	LOCAL CONST Robtarget Tr_meulage_motif_1_P374 :=[[8.13885791015625,-202.05440625,-14.531873046875],[0.696320279376617,-0.571579290814731,-0.275420255163045,0.335527742350052],[0,0,0,0],[8.999999E+09,8.999999E+09,8.999999E+09,8.999999E+09,8.999999E+09,8.999999E+09]];
	LOCAL CONST Robtarget Tr_meulage_motif_1_P375 :=[[8.663193359375,-201.419984375,-15.4485517578125],[0.696320279376617,-0.571579290814731,-0.275420255163045,0.335527742350052],[0,0,0,0],[8.999999E+09,8.999999E+09,8.999999E+09,8.999999E+09,8.999999E+09,8.999999E+09]];
	LOCAL CONST Robtarget Tr_meulage_motif_1_P376 :=[[9.0439765625,-200.94025,-15.87097265625],[0.696320279376617,-0.571579290814731,-0.275420255163045,0.335527742350052],[0,0,0,0],[8.999999E+09,8.999999E+09,8.999999E+09,8.999999E+09,8.999999E+09,8.999999E+09]];
	LOCAL CONST Robtarget Tr_meulage_motif_1_P377 :=[[9.7377255859375,-200.04753125,-16.400830078125],[0.696320279376617,-0.571579290814731,-0.275420255163045,0.335527742350052],[0,0,0,0],[8.999999E+09,8.999999E+09,8.999999E+09,8.999999E+09,8.999999E+09,8.999999E+09]];
	LOCAL CONST Robtarget Tr_meulage_motif_1_P378 :=[[10.2514345703125,-199.37646875,-16.66463671875],[0.696320279376617,-0.571579290814731,-0.275420255163045,0.335527742350052],[0,0,0,0],[8.999999E+09,8.999999E+09,8.999999E+09,8.999999E+09,8.999999E+09,8.999999E+09]];
	LOCAL CONST Robtarget Tr_meulage_motif_1_P379 :=[[10.8147724609375,-198.633921875,-16.868880859375],[0.696320279376617,-0.571579290814731,-0.275420255163045,0.335527742350052],[0,0,0,0],[8.999999E+09,8.999999E+09,8.999999E+09,8.999999E+09,8.999999E+09,8.999999E+09]];
	LOCAL CONST Robtarget Tr_meulage_motif_1_P380 :=[[11.4040810546875,-197.848921875,-16.977291015625],[0.696320279376617,-0.571579290814731,-0.275420255163045,0.335527742350052],[0,0,0,0],[8.999999E+09,8.999999E+09,8.999999E+09,8.999999E+09,8.999999E+09,8.999999E+09]];
	LOCAL CONST Robtarget Tr_meulage_motif_1_P381 :=[[12.000025390625,-197.05515625,-17.087759765625],[0.696320279376617,-0.571579290814731,-0.275420255163045,0.335527742350052],[0,0,0,0],[8.999999E+09,8.999999E+09,8.999999E+09,8.999999E+09,8.999999E+09,8.999999E+09]];
	LOCAL CONST Robtarget Tr_meulage_motif_1_P382 :=[[12.596275390625,-196.252359375,-17.087740234375],[0.696320279376617,-0.571579290814731,-0.275420255163045,0.335527742350052],[0,0,0,0],[8.999999E+09,8.999999E+09,8.999999E+09,8.999999E+09,8.999999E+09,8.999999E+09]];
	LOCAL CONST Robtarget Tr_meulage_motif_1_P383 :=[[13.192525390625,-195.4495625,-17.087720703125],[0.696320279376617,-0.571579290814731,-0.275420255163045,0.335527742350052],[0,0,0,0],[8.999999E+09,8.999999E+09,8.999999E+09,8.999999E+09,8.999999E+09,8.999999E+09]];
	LOCAL CONST Robtarget Tr_meulage_motif_1_P384 :=[[13.7887763671875,-194.646765625,-17.08769921875],[0.696320279376617,-0.571579290814731,-0.275420255163045,0.335527742350052],[0,0,0,0],[8.999999E+09,8.999999E+09,8.999999E+09,8.999999E+09,8.999999E+09,8.999999E+09]];
	LOCAL CONST Robtarget Tr_meulage_motif_1_P385 :=[[14.3850263671875,-193.84396875,-17.0876796875],[0.696320279376617,-0.571579290814731,-0.275420255163045,0.335527742350052],[0,0,0,0],[8.999999E+09,8.999999E+09,8.999999E+09,8.999999E+09,8.999999E+09,8.999999E+09]];
	LOCAL CONST Robtarget Tr_meulage_motif_1_P386 :=[[14.9812763671875,-193.041171875,-17.08766015625],[0.696320279376617,-0.571579290814731,-0.275420255163045,0.335527742350052],[0,0,0,0],[8.999999E+09,8.999999E+09,8.999999E+09,8.999999E+09,8.999999E+09,8.999999E+09]];
	LOCAL CONST Robtarget Tr_meulage_motif_1_P387 :=[[15.57752734375,-192.238375,-17.087638671875],[0.696320279376617,-0.571579290814731,-0.275420255163045,0.335527742350052],[0,0,0,0],[8.999999E+09,8.999999E+09,8.999999E+09,8.999999E+09,8.999999E+09,8.999999E+09]];
	LOCAL CONST Robtarget Tr_meulage_motif_1_P388 :=[[16.17377734375,-191.435578125,-17.087619140625],[0.696320279376617,-0.571579290814731,-0.275420255163045,0.335527742350052],[0,0,0,0],[8.999999E+09,8.999999E+09,8.999999E+09,8.999999E+09,8.999999E+09,8.999999E+09]];
	LOCAL CONST Robtarget Tr_meulage_motif_1_P389 :=[[16.77002734375,-190.632765625,-17.08759765625],[0.696320279376617,-0.571579290814731,-0.275420255163045,0.335527742350052],[0,0,0,0],[8.999999E+09,8.999999E+09,8.999999E+09,8.999999E+09,8.999999E+09,8.999999E+09]];
	LOCAL CONST Robtarget Tr_meulage_motif_1_P390 :=[[17.36627734375,-189.82996875,-17.087578125],[0.696320279376617,-0.571579290814731,-0.275420255163045,0.335527742350052],[0,0,0,0],[8.999999E+09,8.999999E+09,8.999999E+09,8.999999E+09,8.999999E+09,8.999999E+09]];
	LOCAL CONST Robtarget Tr_meulage_motif_1_P391 :=[[17.96252734375,-189.027171875,-17.08755859375],[0.696320279376617,-0.571579290814731,-0.275420255163045,0.335527742350052],[0,0,0,0],[8.999999E+09,8.999999E+09,8.999999E+09,8.999999E+09,8.999999E+09,8.999999E+09]];
	LOCAL CONST Robtarget Tr_meulage_motif_1_P392 :=[[18.558779296875,-188.224375,-17.087537109375],[0.696320279376617,-0.571579290814731,-0.275420255163045,0.335527742350052],[0,0,0,0],[8.999999E+09,8.999999E+09,8.999999E+09,8.999999E+09,8.999999E+09,8.999999E+09]];
	LOCAL CONST Robtarget Tr_meulage_motif_1_P393 :=[[19.155029296875,-187.421578125,-17.087517578125],[0.696320279376617,-0.571579290814731,-0.275420255163045,0.335527742350052],[0,0,0,0],[8.999999E+09,8.999999E+09,8.999999E+09,8.999999E+09,8.999999E+09,8.999999E+09]];
	LOCAL CONST Robtarget Tr_meulage_motif_1_P394 :=[[19.751279296875,-186.61878125,-17.087498046875],[0.696320279376617,-0.571579290814731,-0.275420255163045,0.335527742350052],[0,0,0,0],[8.999999E+09,8.999999E+09,8.999999E+09,8.999999E+09,8.999999E+09,8.999999E+09]];
	LOCAL CONST Robtarget Tr_meulage_motif_1_P395 :=[[20.347529296875,-185.815984375,-17.0874765625],[0.696320279376617,-0.571579290814731,-0.275420255163045,0.335527742350052],[0,0,0,0],[8.999999E+09,8.999999E+09,8.999999E+09,8.999999E+09,8.999999E+09,8.999999E+09]];
	LOCAL CONST Robtarget Tr_meulage_motif_1_P396 :=[[20.943779296875,-185.0131875,-17.08745703125],[0.696320279376617,-0.571579290814731,-0.275420255163045,0.335527742350052],[0,0,0,0],[8.999999E+09,8.999999E+09,8.999999E+09,8.999999E+09,8.999999E+09,8.999999E+09]];
	LOCAL CONST Robtarget Tr_meulage_motif_1_P397 :=[[21.540029296875,-184.210390625,-17.087435546875],[0.696320279376617,-0.571579290814731,-0.275420255163045,0.335527742350052],[0,0,0,0],[8.999999E+09,8.999999E+09,8.999999E+09,8.999999E+09,8.999999E+09,8.999999E+09]];
	LOCAL CONST Robtarget Tr_meulage_motif_1_P398 :=[[22.136279296875,-183.407578125,-17.087416015625],[0.696320279376617,-0.571579290814731,-0.275420255163045,0.335527742350052],[0,0,0,0],[8.999999E+09,8.999999E+09,8.999999E+09,8.999999E+09,8.999999E+09,8.999999E+09]];
	LOCAL CONST Robtarget Tr_meulage_motif_1_P399 :=[[22.73253125,-182.60478125,-17.087396484375],[0.696320279376617,-0.571579290814731,-0.275420255163045,0.335527742350052],[0,0,0,0],[8.999999E+09,8.999999E+09,8.999999E+09,8.999999E+09,8.999999E+09,8.999999E+09]];
	LOCAL CONST Robtarget Tr_meulage_motif_1_P400 :=[[23.32878125,-181.801984375,-17.087375],[0.696320279376617,-0.571579290814731,-0.275420255163045,0.335527742350052],[0,0,0,0],[8.999999E+09,8.999999E+09,8.999999E+09,8.999999E+09,8.999999E+09,8.999999E+09]];
	LOCAL CONST Robtarget Tr_meulage_motif_1_P401 :=[[23.92503125,-180.9991875,-17.08735546875],[0.696320279376617,-0.571579290814731,-0.275420255163045,0.335527742350052],[0,0,0,0],[8.999999E+09,8.999999E+09,8.999999E+09,8.999999E+09,8.999999E+09,8.999999E+09]];
	LOCAL CONST Robtarget Tr_meulage_motif_1_P402 :=[[24.52128125,-180.196390625,-17.0873359375],[0.696320279376617,-0.571579290814731,-0.275420255163045,0.335527742350052],[0,0,0,0],[8.999999E+09,8.999999E+09,8.999999E+09,8.999999E+09,8.999999E+09,8.999999E+09]];
	LOCAL CONST Robtarget Tr_meulage_motif_1_P403 :=[[25.11753125,-179.39359375,-17.087314453125],[0.696320279376617,-0.571579290814731,-0.275420255163045,0.335527742350052],[0,0,0,0],[8.999999E+09,8.999999E+09,8.999999E+09,8.999999E+09,8.999999E+09,8.999999E+09]];
	LOCAL CONST Robtarget Tr_meulage_motif_1_P404 :=[[25.71378125,-178.590796875,-17.087294921875],[0.696320279376617,-0.571579290814731,-0.275420255163045,0.335527742350052],[0,0,0,0],[8.999999E+09,8.999999E+09,8.999999E+09,8.999999E+09,8.999999E+09,8.999999E+09]];
	LOCAL CONST Robtarget Tr_meulage_motif_1_P405 :=[[26.31003125,-177.788,-17.0872734375],[0.696320279376617,-0.571579290814731,-0.275420255163045,0.335527742350052],[0,0,0,0],[8.999999E+09,8.999999E+09,8.999999E+09,8.999999E+09,8.999999E+09,8.999999E+09]];
	LOCAL CONST Robtarget Tr_meulage_motif_1_P406 :=[[26.906283203125,-176.985203125,-17.08725390625],[0.696320279376617,-0.571579290814731,-0.275420255163045,0.335527742350052],[0,0,0,0],[8.999999E+09,8.999999E+09,8.999999E+09,8.999999E+09,8.999999E+09,8.999999E+09]];
	LOCAL CONST Robtarget Tr_meulage_motif_1_P407 :=[[27.502533203125,-176.18240625,-17.087234375],[0.696320279376617,-0.571579290814731,-0.275420255163045,0.335527742350052],[0,0,0,0],[8.999999E+09,8.999999E+09,8.999999E+09,8.999999E+09,8.999999E+09,8.999999E+09]];
	LOCAL CONST Robtarget Tr_meulage_motif_1_P408 :=[[28.098783203125,-175.37959375,-17.087212890625],[0.696320279376617,-0.571579290814731,-0.275420255163045,0.335527742350052],[0,0,0,0],[8.999999E+09,8.999999E+09,8.999999E+09,8.999999E+09,8.999999E+09,8.999999E+09]];
	LOCAL CONST Robtarget Tr_meulage_motif_1_P409 :=[[28.695033203125,-174.576796875,-17.087193359375],[0.696320279376617,-0.571579290814731,-0.275420255163045,0.335527742350052],[0,0,0,0],[8.999999E+09,8.999999E+09,8.999999E+09,8.999999E+09,8.999999E+09,8.999999E+09]];
	LOCAL CONST Robtarget Tr_meulage_motif_1_P410 :=[[29.291283203125,-173.774,-17.087173828125],[0.696320279376617,-0.571579290814731,-0.275420255163045,0.335527742350052],[0,0,0,0],[8.999999E+09,8.999999E+09,8.999999E+09,8.999999E+09,8.999999E+09,8.999999E+09]];
	LOCAL CONST Robtarget Tr_meulage_motif_1_P411 :=[[29.887533203125,-172.971203125,-17.08715234375],[0.696320279376617,-0.571579290814731,-0.275420255163045,0.335527742350052],[0,0,0,0],[8.999999E+09,8.999999E+09,8.999999E+09,8.999999E+09,8.999999E+09,8.999999E+09]];
	LOCAL CONST Robtarget Tr_meulage_motif_1_P412 :=[[30.48378515625,-172.16840625,-17.0871328125],[0.696320279376617,-0.571579290814731,-0.275420255163045,0.335527742350052],[0,0,0,0],[8.999999E+09,8.999999E+09,8.999999E+09,8.999999E+09,8.999999E+09,8.999999E+09]];
	LOCAL CONST Robtarget Tr_meulage_motif_1_P413 :=[[31.08003515625,-171.365609375,-17.087111328125],[0.696320279376617,-0.571579290814731,-0.275420255163045,0.335527742350052],[0,0,0,0],[8.999999E+09,8.999999E+09,8.999999E+09,8.999999E+09,8.999999E+09,8.999999E+09]];
	LOCAL CONST Robtarget Tr_meulage_motif_1_P414 :=[[31.67628515625,-170.5628125,-17.087091796875],[0.696320279376617,-0.571579290814731,-0.275420255163045,0.335527742350052],[0,0,0,0],[8.999999E+09,8.999999E+09,8.999999E+09,8.999999E+09,8.999999E+09,8.999999E+09]];
	LOCAL CONST Robtarget Tr_meulage_motif_1_P415 :=[[32.27253515625,-169.760015625,-17.087072265625],[0.696320279376617,-0.571579290814731,-0.275420255163045,0.335527742350052],[0,0,0,0],[8.999999E+09,8.999999E+09,8.999999E+09,8.999999E+09,8.999999E+09,8.999999E+09]];
	LOCAL CONST Robtarget Tr_meulage_motif_1_P416 :=[[32.86878515625,-168.95721875,-17.08705078125],[0.696320279376617,-0.571579290814731,-0.275420255163045,0.335527742350052],[0,0,0,0],[8.999999E+09,8.999999E+09,8.999999E+09,8.999999E+09,8.999999E+09,8.999999E+09]];
	LOCAL CONST Robtarget Tr_meulage_motif_1_P417 :=[[33.46503515625,-168.15440625,-17.08703125],[0.696320279376617,-0.571579290814731,-0.275420255163045,0.335527742350052],[0,0,0,0],[8.999999E+09,8.999999E+09,8.999999E+09,8.999999E+09,8.999999E+09,8.999999E+09]];
	LOCAL CONST Robtarget Tr_meulage_motif_1_P418 :=[[34.06128515625,-167.351609375,-17.08701171875],[0.696320279376617,-0.571579290814731,-0.275420255163045,0.335527742350052],[0,0,0,0],[8.999999E+09,8.999999E+09,8.999999E+09,8.999999E+09,8.999999E+09,8.999999E+09]];
	LOCAL CONST Robtarget Tr_meulage_motif_1_P419 :=[[34.65753515625,-166.5488125,-17.086990234375],[0.696320279376617,-0.571579290814731,-0.275420255163045,0.335527742350052],[0,0,0,0],[8.999999E+09,8.999999E+09,8.999999E+09,8.999999E+09,8.999999E+09,8.999999E+09]];
	LOCAL CONST Robtarget Tr_meulage_motif_1_P420 :=[[35.25378515625,-165.746015625,-17.086970703125],[0.696320279376617,-0.571579290814731,-0.275420255163045,0.335527742350052],[0,0,0,0],[8.999999E+09,8.999999E+09,8.999999E+09,8.999999E+09,8.999999E+09,8.999999E+09]];
	LOCAL CONST Robtarget Tr_meulage_motif_1_P421 :=[[35.85003515625,-164.94321875,-17.08694921875],[0.696320279376617,-0.571579290814731,-0.275420255163045,0.335527742350052],[0,0,0,0],[8.999999E+09,8.999999E+09,8.999999E+09,8.999999E+09,8.999999E+09,8.999999E+09]];
	LOCAL CONST Robtarget Tr_meulage_motif_1_P422 :=[[36.4462890625,-164.140421875,-17.0869296875],[0.696320279376617,-0.571579290814731,-0.275420255163045,0.335527742350052],[0,0,0,0],[8.999999E+09,8.999999E+09,8.999999E+09,8.999999E+09,8.999999E+09,8.999999E+09]];
	LOCAL CONST Robtarget Tr_meulage_motif_1_P423 :=[[37.0425390625,-163.337625,-17.08691015625],[0.696320279376617,-0.571579290814731,-0.275420255163045,0.335527742350052],[0,0,0,0],[8.999999E+09,8.999999E+09,8.999999E+09,8.999999E+09,8.999999E+09,8.999999E+09]];
	LOCAL CONST Robtarget Tr_meulage_motif_1_P424 :=[[37.6387890625,-162.534828125,-17.086888671875],[0.696320279376617,-0.571579290814731,-0.275420255163045,0.335527742350052],[0,0,0,0],[8.999999E+09,8.999999E+09,8.999999E+09,8.999999E+09,8.999999E+09,8.999999E+09]];
	LOCAL CONST Robtarget Tr_meulage_motif_1_P425 :=[[38.2350390625,-161.73203125,-17.086869140625],[0.696320279376617,-0.571579290814731,-0.275420255163045,0.335527742350052],[0,0,0,0],[8.999999E+09,8.999999E+09,8.999999E+09,8.999999E+09,8.999999E+09,8.999999E+09]];
	LOCAL CONST Robtarget Tr_meulage_motif_1_P426 :=[[38.8312890625,-160.92921875,-17.086849609375],[0.696320279376617,-0.571579290814731,-0.275420255163045,0.335527742350052],[0,0,0,0],[8.999999E+09,8.999999E+09,8.999999E+09,8.999999E+09,8.999999E+09,8.999999E+09]];
	LOCAL CONST Robtarget Tr_meulage_motif_1_P427 :=[[39.4275390625,-160.126421875,-17.086828125],[0.696320279376617,-0.571579290814731,-0.275420255163045,0.335527742350052],[0,0,0,0],[8.999999E+09,8.999999E+09,8.999999E+09,8.999999E+09,8.999999E+09,8.999999E+09]];
	LOCAL CONST Robtarget Tr_meulage_motif_1_P428 :=[[40.0237890625,-159.323625,-17.08680859375],[0.696320279376617,-0.571579290814731,-0.275420255163045,0.335527742350052],[0,0,0,0],[8.999999E+09,8.999999E+09,8.999999E+09,8.999999E+09,8.999999E+09,8.999999E+09]];
	LOCAL CONST Robtarget Tr_meulage_motif_1_P429 :=[[40.6200390625,-158.520828125,-17.086787109375],[0.696320279376617,-0.571579290814731,-0.275420255163045,0.335527742350052],[0,0,0,0],[8.999999E+09,8.999999E+09,8.999999E+09,8.999999E+09,8.999999E+09,8.999999E+09]];
	LOCAL CONST Robtarget Tr_meulage_motif_1_P430 :=[[41.2162890625,-157.71803125,-17.086767578125],[0.696320279376617,-0.571579290814731,-0.275420255163045,0.335527742350052],[0,0,0,0],[8.999999E+09,8.999999E+09,8.999999E+09,8.999999E+09,8.999999E+09,8.999999E+09]];
	LOCAL CONST Robtarget Tr_meulage_motif_1_P431 :=[[41.8125390625,-156.915234375,-17.086748046875],[0.696320279376617,-0.571579290814731,-0.275420255163045,0.335527742350052],[0,0,0,0],[8.999999E+09,8.999999E+09,8.999999E+09,8.999999E+09,8.999999E+09,8.999999E+09]];
	LOCAL CONST Robtarget Tr_meulage_motif_1_P432 :=[[42.4087890625,-156.1124375,-17.0867265625],[0.696320279376617,-0.571579290814731,-0.275420255163045,0.335527742350052],[0,0,0,0],[8.999999E+09,8.999999E+09,8.999999E+09,8.999999E+09,8.999999E+09,8.999999E+09]];
	LOCAL CONST Robtarget Tr_meulage_motif_1_P433 :=[[43.0050390625,-155.309640625,-17.08670703125],[0.696320279376617,-0.571579290814731,-0.275420255163045,0.335527742350052],[0,0,0,0],[8.999999E+09,8.999999E+09,8.999999E+09,8.999999E+09,8.999999E+09,8.999999E+09]];
	LOCAL CONST Robtarget Tr_meulage_motif_1_P434 :=[[43.6012890625,-154.50684375,-17.0866875],[0.696320279376617,-0.571579290814731,-0.275420255163045,0.335527742350052],[0,0,0,0],[8.999999E+09,8.999999E+09,8.999999E+09,8.999999E+09,8.999999E+09,8.999999E+09]];
	LOCAL CONST Robtarget Tr_meulage_motif_1_degg1 :=[[51.2725174233444,-160.618666051073,-19.0355034471531],[0.696320279376617,-0.571579290814731,-0.275420255163045,0.335527742350052],[0,0,0,0],[8.999999E+09,8.999999E+09,8.999999E+09,8.999999E+09,8.999999E+09,8.999999E+09]];
	LOCAL CONST Robtarget Tr_meulage_motif_1_degg2 :=[[197.025856279388,-276.743289771468,-56.063006443061],[0.696320279376617,-0.571579290814731,-0.275420255163045,0.335527742350052],[0,0,0,0],[8.999999E+09,8.999999E+09,8.999999E+09,8.999999E+09,8.999999E+09,8.999999E+09]];
	LOCAL CONST Robtarget Tr_meulage_motif_2_App1 :=[[79.1385711104323,111.598654466444,-198.295056790946],[3.80360857770028E-05,0.00767312788400758,0.0049568441043783,-0.999958274808633],[0,0,0,0],[8.999999E+09,8.999999E+09,8.999999E+09,8.999999E+09,8.999999E+09,8.999999E+09]];
	LOCAL CONST Robtarget Tr_meulage_motif_2_App2 :=[[76.2229758211466,109.715021395197,-8.32676672504532],[3.80360857770028E-05,0.00767312788400758,0.0049568441043783,-0.999958274808633],[0,0,0,0],[8.999999E+09,8.999999E+09,8.999999E+09,8.999999E+09,8.999999E+09,8.999999E+09]];
	LOCAL CONST Robtarget Tr_meulage_motif_2_P0 :=[[76.0695234375,109.6158828125,1.67156433105469],[3.80360857770028E-05,0.00767312788400758,0.0049568441043783,-0.999958274808633],[0,0,0,0],[8.999999E+09,8.999999E+09,8.999999E+09,8.999999E+09,8.999999E+09,8.999999E+09]];
	LOCAL CONST Robtarget Tr_meulage_motif_2_P1 :=[[75.071609375,109.5513046875,1.67191589355469],[3.80360857770028E-05,0.00767312788400758,0.0049568441043783,-0.999958274808633],[0,0,0,0],[8.999999E+09,8.999999E+09,8.999999E+09,8.999999E+09,8.999999E+09,8.999999E+09]];
	LOCAL CONST Robtarget Tr_meulage_motif_2_P2 :=[[74.0736953125,109.4867265625,1.67226745605469],[3.80360857770028E-05,0.00767312788400758,0.0049568441043783,-0.999958274808633],[0,0,0,0],[8.999999E+09,8.999999E+09,8.999999E+09,8.999999E+09,8.999999E+09,8.999999E+09]];
	LOCAL CONST Robtarget Tr_meulage_motif_2_P3 :=[[73.07578125,109.4221484375,1.67261889648438],[3.80360857770028E-05,0.00767312788400758,0.0049568441043783,-0.999958274808633],[0,0,0,0],[8.999999E+09,8.999999E+09,8.999999E+09,8.999999E+09,8.999999E+09,8.999999E+09]];
	LOCAL CONST Robtarget Tr_meulage_motif_2_P4 :=[[72.0778671875,109.3575703125,1.67297045898438],[3.80360857770028E-05,0.00767312788400758,0.0049568441043783,-0.999958274808633],[0,0,0,0],[8.999999E+09,8.999999E+09,8.999999E+09,8.999999E+09,8.999999E+09,8.999999E+09]];
	LOCAL CONST Robtarget Tr_meulage_motif_2_P5 :=[[71.079953125,109.293,1.67332202148438],[3.80360857770028E-05,0.00767312788400758,0.0049568441043783,-0.999958274808633],[0,0,0,0],[8.999999E+09,8.999999E+09,8.999999E+09,8.999999E+09,8.999999E+09,8.999999E+09]];
	LOCAL CONST Robtarget Tr_meulage_motif_2_P6 :=[[70.082046875,109.228421875,1.67367358398438],[3.80360857770028E-05,0.00767312788400758,0.0049568441043783,-0.999958274808633],[0,0,0,0],[8.999999E+09,8.999999E+09,8.999999E+09,8.999999E+09,8.999999E+09,8.999999E+09]];
	LOCAL CONST Robtarget Tr_meulage_motif_2_P7 :=[[69.0841328125,109.16384375,1.67402514648437],[3.80360857770028E-05,0.00767312788400758,0.0049568441043783,-0.999958274808633],[0,0,0,0],[8.999999E+09,8.999999E+09,8.999999E+09,8.999999E+09,8.999999E+09,8.999999E+09]];
	LOCAL CONST Robtarget Tr_meulage_motif_2_P8 :=[[68.08621875,109.099265625,1.67437670898438],[3.80360857770028E-05,0.00767312788400758,0.0049568441043783,-0.999958274808633],[0,0,0,0],[8.999999E+09,8.999999E+09,8.999999E+09,8.999999E+09,8.999999E+09,8.999999E+09]];
	LOCAL CONST Robtarget Tr_meulage_motif_2_P9 :=[[67.0883046875,109.0346875,1.67472827148437],[3.80360857770028E-05,0.00767312788400758,0.0049568441043783,-0.999958274808633],[0,0,0,0],[8.999999E+09,8.999999E+09,8.999999E+09,8.999999E+09,8.999999E+09,8.999999E+09]];
	LOCAL CONST Robtarget Tr_meulage_motif_2_P10 :=[[66.090390625,108.9701171875,1.67507983398438],[3.80360857770028E-05,0.00767312788400758,0.0049568441043783,-0.999958274808633],[0,0,0,0],[8.999999E+09,8.999999E+09,8.999999E+09,8.999999E+09,8.999999E+09,8.999999E+09]];
	LOCAL CONST Robtarget Tr_meulage_motif_2_P11 :=[[65.09248046875,108.9055390625,1.67543127441406],[3.80360857770028E-05,0.00767312788400758,0.0049568441043783,-0.999958274808633],[0,0,0,0],[8.999999E+09,8.999999E+09,8.999999E+09,8.999999E+09,8.999999E+09,8.999999E+09]];
	LOCAL CONST Robtarget Tr_meulage_motif_2_P12 :=[[64.09456640625,108.8409609375,1.67578283691406],[3.80360857770028E-05,0.00767312788400758,0.0049568441043783,-0.999958274808633],[0,0,0,0],[8.999999E+09,8.999999E+09,8.999999E+09,8.999999E+09,8.999999E+09,8.999999E+09]];
	LOCAL CONST Robtarget Tr_meulage_motif_2_P13 :=[[63.09665625,108.7763828125,1.67613439941406],[3.80360857770028E-05,0.00767312788400758,0.0049568441043783,-0.999958274808633],[0,0,0,0],[8.999999E+09,8.999999E+09,8.999999E+09,8.999999E+09,8.999999E+09,8.999999E+09]];
	LOCAL CONST Robtarget Tr_meulage_motif_2_P14 :=[[62.0987421875,108.7118046875,1.67648596191406],[3.80360857770028E-05,0.00767312788400758,0.0049568441043783,-0.999958274808633],[0,0,0,0],[8.999999E+09,8.999999E+09,8.999999E+09,8.999999E+09,8.999999E+09,8.999999E+09]];
	LOCAL CONST Robtarget Tr_meulage_motif_2_P15 :=[[61.100828125,108.6472265625,1.67683752441406],[3.80360857770028E-05,0.00767312788400758,0.0049568441043783,-0.999958274808633],[0,0,0,0],[8.999999E+09,8.999999E+09,8.999999E+09,8.999999E+09,8.999999E+09,8.999999E+09]];
	LOCAL CONST Robtarget Tr_meulage_motif_2_P16 :=[[60.10291796875,108.58265625,1.67718908691406],[3.80360857770028E-05,0.00767312788400758,0.0049568441043783,-0.999958274808633],[0,0,0,0],[8.999999E+09,8.999999E+09,8.999999E+09,8.999999E+09,8.999999E+09,8.999999E+09]];
	LOCAL CONST Robtarget Tr_meulage_motif_2_P17 :=[[59.10500390625,108.518078125,1.67754064941406],[3.80360857770028E-05,0.00767312788400758,0.0049568441043783,-0.999958274808633],[0,0,0,0],[8.999999E+09,8.999999E+09,8.999999E+09,8.999999E+09,8.999999E+09,8.999999E+09]];
	LOCAL CONST Robtarget Tr_meulage_motif_2_P18 :=[[58.10708984375,108.4535,1.67789221191406],[3.80360857770028E-05,0.00767312788400758,0.0049568441043783,-0.999958274808633],[0,0,0,0],[8.999999E+09,8.999999E+09,8.999999E+09,8.999999E+09,8.999999E+09,8.999999E+09]];
	LOCAL CONST Robtarget Tr_meulage_motif_2_P19 :=[[57.1094609375,108.499765625,1.67763696289063],[3.80360857770028E-05,0.00767312788400758,0.0049568441043783,-0.999958274808633],[0,0,0,0],[8.999999E+09,8.999999E+09,8.999999E+09,8.999999E+09,8.999999E+09,8.999999E+09]];
	LOCAL CONST Robtarget Tr_meulage_motif_2_P20 :=[[56.151296875,108.649390625,1.67681604003906],[3.80360857770028E-05,0.00767312788400758,0.0049568441043783,-0.999958274808633],[0,0,0,0],[8.999999E+09,8.999999E+09,8.999999E+09,8.999999E+09,8.999999E+09,8.999999E+09]];
	LOCAL CONST Robtarget Tr_meulage_motif_2_P21 :=[[55.2828046875,108.86559375,1.675630859375],[3.80360857770028E-05,0.00767312788400758,0.0049568441043783,-0.999958274808633],[0,0,0,0],[8.999999E+09,8.999999E+09,8.999999E+09,8.999999E+09,8.999999E+09,8.999999E+09]];
	LOCAL CONST Robtarget Tr_meulage_motif_2_P22 :=[[54.51661328125,109.0925234375,1.67438720703125],[3.80360857770028E-05,0.00767312788400758,0.0049568441043783,-0.999958274808633],[0,0,0,0],[8.999999E+09,8.999999E+09,8.999999E+09,8.999999E+09,8.999999E+09,8.999999E+09]];
	LOCAL CONST Robtarget Tr_meulage_motif_2_P23 :=[[53.37805859375,109.63625,1.67140869140625],[3.80360857770028E-05,0.00767312788400758,0.0049568441043783,-0.999958274808633],[0,0,0,0],[8.999999E+09,8.999999E+09,8.999999E+09,8.999999E+09,8.999999E+09,8.999999E+09]];
	LOCAL CONST Robtarget Tr_meulage_motif_2_P24 :=[[52.30158203125,110.4160078125,1.66713830566406],[3.80360857770028E-05,0.00767312788400758,0.0049568441043783,-0.999958274808633],[0,0,0,0],[8.999999E+09,8.999999E+09,8.999999E+09,8.999999E+09,8.999999E+09,8.999999E+09]];
	LOCAL CONST Robtarget Tr_meulage_motif_2_P25 :=[[51.38957421875,111.3829921875,1.66184338378906],[3.80360857770028E-05,0.00767312788400758,0.0049568441043783,-0.999958274808633],[0,0,0,0],[8.999999E+09,8.999999E+09,8.999999E+09,8.999999E+09,8.999999E+09,8.999999E+09]];
	LOCAL CONST Robtarget Tr_meulage_motif_2_P26 :=[[50.830359375,112.4653046875,1.65591772460938],[3.80360857770028E-05,0.00767312788400758,0.0049568441043783,-0.999958274808633],[0,0,0,0],[8.999999E+09,8.999999E+09,8.999999E+09,8.999999E+09,8.999999E+09,8.999999E+09]];
	LOCAL CONST Robtarget Tr_meulage_motif_2_P27 :=[[50.75840625,113.1580625,1.65212561035156],[3.80360857770028E-05,0.00767312788400758,0.0049568441043783,-0.999958274808633],[0,0,0,0],[8.999999E+09,8.999999E+09,8.999999E+09,8.999999E+09,8.999999E+09,8.999999E+09]];
	LOCAL CONST Robtarget Tr_meulage_motif_2_P28 :=[[50.71570703125,113.817921875,1.64851342773437],[3.80360857770028E-05,0.00767312788400758,0.0049568441043783,-0.999958274808633],[0,0,0,0],[8.999999E+09,8.999999E+09,8.999999E+09,8.999999E+09,8.999999E+09,8.999999E+09]];
	LOCAL CONST Robtarget Tr_meulage_motif_2_P29 :=[[50.7277734375,114.481171875,1.64488293457031],[3.80360857770028E-05,0.00767312788400758,0.0049568441043783,-0.999958274808633],[0,0,0,0],[8.999999E+09,8.999999E+09,8.999999E+09,8.999999E+09,8.999999E+09,8.999999E+09]];
	LOCAL CONST Robtarget Tr_meulage_motif_2_P30 :=[[51.1538046875,115.61278125,1.638689453125],[3.80360857770028E-05,0.00767312788400758,0.0049568441043783,-0.999958274808633],[0,0,0,0],[8.999999E+09,8.999999E+09,8.999999E+09,8.999999E+09,8.999999E+09,8.999999E+09]];
	LOCAL CONST Robtarget Tr_meulage_motif_2_P31 :=[[51.94363671875,116.672609375,1.6328896484375],[3.80360857770028E-05,0.00767312788400758,0.0049568441043783,-0.999958274808633],[0,0,0,0],[8.999999E+09,8.999999E+09,8.999999E+09,8.999999E+09,8.999999E+09,8.999999E+09]];
	LOCAL CONST Robtarget Tr_meulage_motif_2_P32 :=[[52.91137890625,117.565828125,1.62800207519531],[3.80360857770028E-05,0.00767312788400758,0.0049568441043783,-0.999958274808633],[0,0,0,0],[8.999999E+09,8.999999E+09,8.999999E+09,8.999999E+09,8.999999E+09,8.999999E+09]];
	LOCAL CONST Robtarget Tr_meulage_motif_2_P33 :=[[53.571484375,118.0051171875,1.62559875488281],[3.80360857770028E-05,0.00767312788400758,0.0049568441043783,-0.999958274808633],[0,0,0,0],[8.999999E+09,8.999999E+09,8.999999E+09,8.999999E+09,8.999999E+09,8.999999E+09]];
	LOCAL CONST Robtarget Tr_meulage_motif_2_P34 :=[[54.69573828125,118.5664140625,1.62252844238281],[3.80360857770028E-05,0.00767312788400758,0.0049568441043783,-0.999958274808633],[0,0,0,0],[8.999999E+09,8.999999E+09,8.999999E+09,8.999999E+09,8.999999E+09,8.999999E+09]];
	LOCAL CONST Robtarget Tr_meulage_motif_2_P35 :=[[55.52194921875,118.884515625,1.62078881835938],[3.80360857770028E-05,0.00767312788400758,0.0049568441043783,-0.999958274808633],[0,0,0,0],[8.999999E+09,8.999999E+09,8.999999E+09,8.999999E+09,8.999999E+09,8.999999E+09]];
	LOCAL CONST Robtarget Tr_meulage_motif_2_P36 :=[[56.43880078125,119.1487421875,1.61934423828125],[3.80360857770028E-05,0.00767312788400758,0.0049568441043783,-0.999958274808633],[0,0,0,0],[8.999999E+09,8.999999E+09,8.999999E+09,8.999999E+09,8.999999E+09,8.999999E+09]];
	LOCAL CONST Robtarget Tr_meulage_motif_2_P37 :=[[57.41130078125,119.3204921875,1.61840600585937],[3.80360857770028E-05,0.00767312788400758,0.0049568441043783,-0.999958274808633],[0,0,0,0],[8.999999E+09,8.999999E+09,8.999999E+09,8.999999E+09,8.999999E+09,8.999999E+09]];
	LOCAL CONST Robtarget Tr_meulage_motif_2_P38 :=[[58.39465234375,119.494953125,1.61745288085938],[3.80360857770028E-05,0.00767312788400758,0.0049568441043783,-0.999958274808633],[0,0,0,0],[8.999999E+09,8.999999E+09,8.999999E+09,8.999999E+09,8.999999E+09,8.999999E+09]];
	LOCAL CONST Robtarget Tr_meulage_motif_2_P39 :=[[59.3925625,119.55953125,1.61710131835937],[3.80360857770028E-05,0.00767312788400758,0.0049568441043783,-0.999958274808633],[0,0,0,0],[8.999999E+09,8.999999E+09,8.999999E+09,8.999999E+09,8.999999E+09,8.999999E+09]];
	LOCAL CONST Robtarget Tr_meulage_motif_2_P40 :=[[60.3904765625,119.624109375,1.61674975585938],[3.80360857770028E-05,0.00767312788400758,0.0049568441043783,-0.999958274808633],[0,0,0,0],[8.999999E+09,8.999999E+09,8.999999E+09,8.999999E+09,8.999999E+09,8.999999E+09]];
	LOCAL CONST Robtarget Tr_meulage_motif_2_P41 :=[[61.388390625,119.6886796875,1.61639819335937],[3.80360857770028E-05,0.00767312788400758,0.0049568441043783,-0.999958274808633],[0,0,0,0],[8.999999E+09,8.999999E+09,8.999999E+09,8.999999E+09,8.999999E+09,8.999999E+09]];
	LOCAL CONST Robtarget Tr_meulage_motif_2_P42 :=[[62.38630078125,119.7532578125,1.61604675292969],[3.80360857770028E-05,0.00767312788400758,0.0049568441043783,-0.999958274808633],[0,0,0,0],[8.999999E+09,8.999999E+09,8.999999E+09,8.999999E+09,8.999999E+09,8.999999E+09]];
	LOCAL CONST Robtarget Tr_meulage_motif_2_P43 :=[[63.38421484375,119.8178359375,1.61569519042969],[3.80360857770028E-05,0.00767312788400758,0.0049568441043783,-0.999958274808633],[0,0,0,0],[8.999999E+09,8.999999E+09,8.999999E+09,8.999999E+09,8.999999E+09,8.999999E+09]];
	LOCAL CONST Robtarget Tr_meulage_motif_2_P44 :=[[64.38212890625,119.8824140625,1.61534362792969],[3.80360857770028E-05,0.00767312788400758,0.0049568441043783,-0.999958274808633],[0,0,0,0],[8.999999E+09,8.999999E+09,8.999999E+09,8.999999E+09,8.999999E+09,8.999999E+09]];
	LOCAL CONST Robtarget Tr_meulage_motif_2_P45 :=[[65.3800390625,119.9469921875,1.61499206542969],[3.80360857770028E-05,0.00767312788400758,0.0049568441043783,-0.999958274808633],[0,0,0,0],[8.999999E+09,8.999999E+09,8.999999E+09,8.999999E+09,8.999999E+09,8.999999E+09]];
	LOCAL CONST Robtarget Tr_meulage_motif_2_P46 :=[[66.377953125,120.0115625,1.61464050292969],[3.80360857770028E-05,0.00767312788400758,0.0049568441043783,-0.999958274808633],[0,0,0,0],[8.999999E+09,8.999999E+09,8.999999E+09,8.999999E+09,8.999999E+09,8.999999E+09]];
	LOCAL CONST Robtarget Tr_meulage_motif_2_P47 :=[[67.3758671875,120.076140625,1.61428894042969],[3.80360857770028E-05,0.00767312788400758,0.0049568441043783,-0.999958274808633],[0,0,0,0],[8.999999E+09,8.999999E+09,8.999999E+09,8.999999E+09,8.999999E+09,8.999999E+09]];
	LOCAL CONST Robtarget Tr_meulage_motif_2_P48 :=[[68.37378125,120.14071875,1.61393737792969],[3.80360857770028E-05,0.00767312788400758,0.0049568441043783,-0.999958274808633],[0,0,0,0],[8.999999E+09,8.999999E+09,8.999999E+09,8.999999E+09,8.999999E+09,8.999999E+09]];
	LOCAL CONST Robtarget Tr_meulage_motif_2_P49 :=[[69.357125,120.3151796875,1.612984375],[3.80360857770028E-05,0.00767312788400758,0.0049568441043783,-0.999958274808633],[0,0,0,0],[8.999999E+09,8.999999E+09,8.999999E+09,8.999999E+09,8.999999E+09,8.999999E+09]];
	LOCAL CONST Robtarget Tr_meulage_motif_2_P50 :=[[70.288015625,120.5870390625,1.611498046875],[3.80360857770028E-05,0.00767312788400758,0.0049568441043783,-0.999958274808633],[0,0,0,0],[8.999999E+09,8.999999E+09,8.999999E+09,8.999999E+09,8.999999E+09,8.999999E+09]];
	LOCAL CONST Robtarget Tr_meulage_motif_2_P51 :=[[71.1213984375,120.9133828125,1.60971325683594],[3.80360857770028E-05,0.00767312788400758,0.0049568441043783,-0.999958274808633],[0,0,0,0],[8.999999E+09,8.999999E+09,8.999999E+09,8.999999E+09,8.999999E+09,8.999999E+09]];
	LOCAL CONST Robtarget Tr_meulage_motif_2_P52 :=[[71.8117734375,121.26284375,1.6078017578125],[3.80360857770028E-05,0.00767312788400758,0.0049568441043783,-0.999958274808633],[0,0,0,0],[8.999999E+09,8.999999E+09,8.999999E+09,8.999999E+09,8.999999E+09,8.999999E+09]];
	LOCAL CONST Robtarget Tr_meulage_motif_2_P53 :=[[72.801296875,121.99078125,1.60381896972656],[3.80360857770028E-05,0.00767312788400758,0.0049568441043783,-0.999958274808633],[0,0,0,0],[8.999999E+09,8.999999E+09,8.999999E+09,8.999999E+09,8.999999E+09,8.999999E+09]];
	LOCAL CONST Robtarget Tr_meulage_motif_2_P54 :=[[73.6431015625,122.9490703125,1.59857507324219],[3.80360857770028E-05,0.00767312788400758,0.0049568441043783,-0.999958274808633],[0,0,0,0],[8.999999E+09,8.999999E+09,8.999999E+09,8.999999E+09,8.999999E+09,8.999999E+09]];
	LOCAL CONST Robtarget Tr_meulage_motif_2_P55 :=[[74.10940625,124.0274453125,1.59267297363281],[3.80360857770028E-05,0.00767312788400758,0.0049568441043783,-0.999958274808633],[0,0,0,0],[8.999999E+09,8.999999E+09,8.999999E+09,8.999999E+09,8.999999E+09,8.999999E+09]];
	LOCAL CONST Robtarget Tr_meulage_motif_2_P56 :=[[74.2490390625,124.731140625,1.5888212890625],[3.80360857770028E-05,0.00767312788400758,0.0049568441043783,-0.999958274808633],[0,0,0,0],[8.999999E+09,8.999999E+09,8.999999E+09,8.999999E+09,8.999999E+09,8.999999E+09]];
	LOCAL CONST Robtarget Tr_meulage_motif_2_P57 :=[[74.2630234375,125.5036484375,1.5845927734375],[3.80360857770028E-05,0.00767312788400758,0.0049568441043783,-0.999958274808633],[0,0,0,0],[8.999999E+09,8.999999E+09,8.999999E+09,8.999999E+09,8.999999E+09,8.999999E+09]];
	LOCAL CONST Robtarget Tr_meulage_motif_2_P58 :=[[74.1465078125,126.267578125,1.58041076660156],[3.80360857770028E-05,0.00767312788400758,0.0049568441043783,-0.999958274808633],[0,0,0,0],[8.999999E+09,8.999999E+09,8.999999E+09,8.999999E+09,8.999999E+09,8.999999E+09]];
	LOCAL CONST Robtarget Tr_meulage_motif_2_P59 :=[[73.65621875,127.34640625,1.57450451660156],[3.80360857770028E-05,0.00767312788400758,0.0049568441043783,-0.999958274808633],[0,0,0,0],[8.999999E+09,8.999999E+09,8.999999E+09,8.999999E+09,8.999999E+09,8.999999E+09]];
	LOCAL CONST Robtarget Tr_meulage_motif_2_P60 :=[[73.204953125,127.9041015625,1.57145080566406],[3.80360857770028E-05,0.00767312788400758,0.0049568441043783,-0.999958274808633],[0,0,0,0],[8.999999E+09,8.999999E+09,8.999999E+09,8.999999E+09,8.999999E+09,8.999999E+09]];
	LOCAL CONST Robtarget Tr_meulage_motif_2_P61 :=[[72.262390625,128.732078125,1.56691674804688],[3.80360857770028E-05,0.00767312788400758,0.0049568441043783,-0.999958274808633],[0,0,0,0],[8.999999E+09,8.999999E+09,8.999999E+09,8.999999E+09,8.999999E+09,8.999999E+09]];
	LOCAL CONST Robtarget Tr_meulage_motif_2_P62 :=[[71.651171875,129.1076953125,1.564859375],[3.80360857770028E-05,0.00767312788400758,0.0049568441043783,-0.999958274808633],[0,0,0,0],[8.999999E+09,8.999999E+09,8.999999E+09,8.999999E+09,8.999999E+09,8.999999E+09]];
	LOCAL CONST Robtarget Tr_meulage_motif_2_P63 :=[[70.5004609375,129.578453125,1.5622802734375],[3.80360857770028E-05,0.00767312788400758,0.0049568441043783,-0.999958274808633],[0,0,0,0],[8.999999E+09,8.999999E+09,8.999999E+09,8.999999E+09,8.999999E+09,8.999999E+09]];
	LOCAL CONST Robtarget Tr_meulage_motif_2_P64 :=[[69.6575078125,129.8200234375,1.56095642089844],[3.80360857770028E-05,0.00767312788400758,0.0049568441043783,-0.999958274808633],[0,0,0,0],[8.999999E+09,8.999999E+09,8.999999E+09,8.999999E+09,8.999999E+09,8.999999E+09]];
	LOCAL CONST Robtarget Tr_meulage_motif_2_P65 :=[[68.71425,129.963875,1.56016711425781],[3.80360857770028E-05,0.00767312788400758,0.0049568441043783,-0.999958274808633],[0,0,0,0],[8.999999E+09,8.999999E+09,8.999999E+09,8.999999E+09,8.999999E+09,8.999999E+09]];
	LOCAL CONST Robtarget Tr_meulage_motif_2_P66 :=[[67.72771875,130.0088515625,1.5599189453125],[3.80360857770028E-05,0.00767312788400758,0.0049568441043783,-0.999958274808633],[0,0,0,0],[8.999999E+09,8.999999E+09,8.999999E+09,8.999999E+09,8.999999E+09,8.999999E+09]];
	LOCAL CONST Robtarget Tr_meulage_motif_2_P67 :=[[66.7300859375,130.0551171875,1.55966381835937],[3.80360857770028E-05,0.00767312788400758,0.0049568441043783,-0.999958274808633],[0,0,0,0],[8.999999E+09,8.999999E+09,8.999999E+09,8.999999E+09,8.999999E+09,8.999999E+09]];
	LOCAL CONST Robtarget Tr_meulage_motif_2_P68 :=[[65.7321796875,129.9905390625,1.56001538085938],[3.80360857770028E-05,0.00767312788400758,0.0049568441043783,-0.999958274808633],[0,0,0,0],[8.999999E+09,8.999999E+09,8.999999E+09,8.999999E+09,8.999999E+09,8.999999E+09]];
	LOCAL CONST Robtarget Tr_meulage_motif_2_P69 :=[[64.734265625,129.92596875,1.56036682128906],[3.80360857770028E-05,0.00767312788400758,0.0049568441043783,-0.999958274808633],[0,0,0,0],[8.999999E+09,8.999999E+09,8.999999E+09,8.999999E+09,8.999999E+09,8.999999E+09]];
	LOCAL CONST Robtarget Tr_meulage_motif_2_P70 :=[[63.7363515625,129.861390625,1.56071838378906],[3.80360857770028E-05,0.00767312788400758,0.0049568441043783,-0.999958274808633],[0,0,0,0],[8.999999E+09,8.999999E+09,8.999999E+09,8.999999E+09,8.999999E+09,8.999999E+09]];
	LOCAL CONST Robtarget Tr_meulage_motif_2_P71 :=[[62.7384375,129.7968125,1.56106994628906],[3.80360857770028E-05,0.00767312788400758,0.0049568441043783,-0.999958274808633],[0,0,0,0],[8.999999E+09,8.999999E+09,8.999999E+09,8.999999E+09,8.999999E+09,8.999999E+09]];
	LOCAL CONST Robtarget Tr_meulage_motif_2_P72 :=[[61.74052734375,129.732234375,1.56142150878906],[3.80360857770028E-05,0.00767312788400758,0.0049568441043783,-0.999958274808633],[0,0,0,0],[8.999999E+09,8.999999E+09,8.999999E+09,8.999999E+09,8.999999E+09,8.999999E+09]];
	LOCAL CONST Robtarget Tr_meulage_motif_2_P73 :=[[60.74261328125,129.66765625,1.56177307128906],[3.80360857770028E-05,0.00767312788400758,0.0049568441043783,-0.999958274808633],[0,0,0,0],[8.999999E+09,8.999999E+09,8.999999E+09,8.999999E+09,8.999999E+09,8.999999E+09]];
	LOCAL CONST Robtarget Tr_meulage_motif_2_P74 :=[[59.74469921875,129.6030859375,1.56212463378906],[3.80360857770028E-05,0.00767312788400758,0.0049568441043783,-0.999958274808633],[0,0,0,0],[8.999999E+09,8.999999E+09,8.999999E+09,8.999999E+09,8.999999E+09,8.999999E+09]];
	LOCAL CONST Robtarget Tr_meulage_motif_2_P75 :=[[58.7467890625,129.5385078125,1.56247619628906],[3.80360857770028E-05,0.00767312788400758,0.0049568441043783,-0.999958274808633],[0,0,0,0],[8.999999E+09,8.999999E+09,8.999999E+09,8.999999E+09,8.999999E+09,8.999999E+09]];
	LOCAL CONST Robtarget Tr_meulage_motif_2_P76 :=[[57.748875,129.4739296875,1.56282775878906],[3.80360857770028E-05,0.00767312788400758,0.0049568441043783,-0.999958274808633],[0,0,0,0],[8.999999E+09,8.999999E+09,8.999999E+09,8.999999E+09,8.999999E+09,8.999999E+09]];
	LOCAL CONST Robtarget Tr_meulage_motif_2_P77 :=[[56.75096484375,129.4093515625,1.56317919921875],[3.80360857770028E-05,0.00767312788400758,0.0049568441043783,-0.999958274808633],[0,0,0,0],[8.999999E+09,8.999999E+09,8.999999E+09,8.999999E+09,8.999999E+09,8.999999E+09]];
	LOCAL CONST Robtarget Tr_meulage_motif_2_P78 :=[[55.75333203125,129.4556171875,1.56292407226563],[3.80360857770028E-05,0.00767312788400758,0.0049568441043783,-0.999958274808633],[0,0,0,0],[8.999999E+09,8.999999E+09,8.999999E+09,8.999999E+09,8.999999E+09,8.999999E+09]];
	LOCAL CONST Robtarget Tr_meulage_motif_2_P79 :=[[54.79516796875,129.6052421875,1.56210314941406],[3.80360857770028E-05,0.00767312788400758,0.0049568441043783,-0.999958274808633],[0,0,0,0],[8.999999E+09,8.999999E+09,8.999999E+09,8.999999E+09,8.999999E+09,8.999999E+09]];
	LOCAL CONST Robtarget Tr_meulage_motif_2_P80 :=[[53.92667578125,129.8214453125,1.56091796875],[3.80360857770028E-05,0.00767312788400758,0.0049568441043783,-0.999958274808633],[0,0,0,0],[8.999999E+09,8.999999E+09,8.999999E+09,8.999999E+09,8.999999E+09,8.999999E+09]];
	LOCAL CONST Robtarget Tr_meulage_motif_2_P81 :=[[53.160484375,130.048375,1.55967431640625],[3.80360857770028E-05,0.00767312788400758,0.0049568441043783,-0.999958274808633],[0,0,0,0],[8.999999E+09,8.999999E+09,8.999999E+09,8.999999E+09,8.999999E+09,8.999999E+09]];
	LOCAL CONST Robtarget Tr_meulage_motif_2_P82 :=[[52.0219296875,130.5921015625,1.55669580078125],[3.80360857770028E-05,0.00767312788400758,0.0049568441043783,-0.999958274808633],[0,0,0,0],[8.999999E+09,8.999999E+09,8.999999E+09,8.999999E+09,8.999999E+09,8.999999E+09]];
	LOCAL CONST Robtarget Tr_meulage_motif_2_P83 :=[[51.0094765625,131.42240625,1.55214880371094],[3.80360857770028E-05,0.00767312788400758,0.0049568441043783,-0.999958274808633],[0,0,0,0],[8.999999E+09,8.999999E+09,8.999999E+09,8.999999E+09,8.999999E+09,8.999999E+09]];
	LOCAL CONST Robtarget Tr_meulage_motif_2_P84 :=[[50.3314921875,132.466796875,1.5464306640625],[3.80360857770028E-05,0.00767312788400758,0.0049568441043783,-0.999958274808633],[0,0,0,0],[8.999999E+09,8.999999E+09,8.999999E+09,8.999999E+09,8.999999E+09,8.999999E+09]];
	LOCAL CONST Robtarget Tr_meulage_motif_2_P85 :=[[50.09896484375,133.43815625,1.54111303710938],[3.80360857770028E-05,0.00767312788400758,0.0049568441043783,-0.999958274808633],[0,0,0,0],[8.999999E+09,8.999999E+09,8.999999E+09,8.999999E+09,8.999999E+09,8.999999E+09]];
	LOCAL CONST Robtarget Tr_meulage_motif_2_P86 :=[[50.2169453125,133.650875,1.53994885253906],[3.80360857770028E-05,0.00767312788400758,0.0049568441043783,-0.999958274808633],[0,0,0,0],[8.999999E+09,8.999999E+09,8.999999E+09,8.999999E+09,8.999999E+09,8.999999E+09]];
	LOCAL CONST Robtarget Tr_meulage_motif_2_P87 :=[[50.29315234375,134.38371875,1.5359375],[3.80360857770028E-05,0.00767312788400758,0.0049568441043783,-0.999958274808633],[0,0,0,0],[8.999999E+09,8.999999E+09,8.999999E+09,8.999999E+09,8.999999E+09,8.999999E+09]];
	LOCAL CONST Robtarget Tr_meulage_motif_2_P88 :=[[50.91522265625,135.362828125,1.5305791015625],[3.80360857770028E-05,0.00767312788400758,0.0049568441043783,-0.999958274808633],[0,0,0,0],[8.999999E+09,8.999999E+09,8.999999E+09,8.999999E+09,8.999999E+09,8.999999E+09]];
	LOCAL CONST Robtarget Tr_meulage_motif_2_P89 :=[[51.44173046875,135.8616875,1.52784948730469],[3.80360857770028E-05,0.00767312788400758,0.0049568441043783,-0.999958274808633],[0,0,0,0],[8.999999E+09,8.999999E+09,8.999999E+09,8.999999E+09,8.999999E+09,8.999999E+09]];
	LOCAL CONST Robtarget Tr_meulage_motif_2_P90 :=[[52.5354296875,136.464,1.5245546875],[3.80360857770028E-05,0.00767312788400758,0.0049568441043783,-0.999958274808633],[0,0,0,0],[8.999999E+09,8.999999E+09,8.999999E+09,8.999999E+09,8.999999E+09,8.999999E+09]];
	LOCAL CONST Robtarget Tr_meulage_motif_2_P91 :=[[53.361640625,136.782109375,1.52281494140625],[3.80360857770028E-05,0.00767312788400758,0.0049568441043783,-0.999958274808633],[0,0,0,0],[8.999999E+09,8.999999E+09,8.999999E+09,8.999999E+09,8.999999E+09,8.999999E+09]];
	LOCAL CONST Robtarget Tr_meulage_motif_2_P92 :=[[54.2784921875,137.046328125,1.52137036132813],[3.80360857770028E-05,0.00767312788400758,0.0049568441043783,-0.999958274808633],[0,0,0,0],[8.999999E+09,8.999999E+09,8.999999E+09,8.999999E+09,8.999999E+09,8.999999E+09]];
	LOCAL CONST Robtarget Tr_meulage_motif_2_P93 :=[[55.2509921875,137.218078125,1.52043212890625],[3.80360857770028E-05,0.00767312788400758,0.0049568441043783,-0.999958274808633],[0,0,0,0],[8.999999E+09,8.999999E+09,8.999999E+09,8.999999E+09,8.999999E+09,8.999999E+09]];
	LOCAL CONST Robtarget Tr_meulage_motif_2_P94 :=[[56.23434375,137.39253125,1.51947912597656],[3.80360857770028E-05,0.00767312788400758,0.0049568441043783,-0.999958274808633],[0,0,0,0],[8.999999E+09,8.999999E+09,8.999999E+09,8.999999E+09,8.999999E+09,8.999999E+09]];
	LOCAL CONST Robtarget Tr_meulage_motif_2_P95 :=[[57.23225390625,137.457109375,1.51912756347656],[3.80360857770028E-05,0.00767312788400758,0.0049568441043783,-0.999958274808633],[0,0,0,0],[8.999999E+09,8.999999E+09,8.999999E+09,8.999999E+09,8.999999E+09,8.999999E+09]];
	LOCAL CONST Robtarget Tr_meulage_motif_2_P96 :=[[58.23016796875,137.5216875,1.51877600097656],[3.80360857770028E-05,0.00767312788400758,0.0049568441043783,-0.999958274808633],[0,0,0,0],[8.999999E+09,8.999999E+09,8.999999E+09,8.999999E+09,8.999999E+09,8.999999E+09]];
	LOCAL CONST Robtarget Tr_meulage_motif_2_P97 :=[[59.22808203125,137.586265625,1.51842443847656],[3.80360857770028E-05,0.00767312788400758,0.0049568441043783,-0.999958274808633],[0,0,0,0],[8.999999E+09,8.999999E+09,8.999999E+09,8.999999E+09,8.999999E+09,8.999999E+09]];
	LOCAL CONST Robtarget Tr_meulage_motif_2_P98 :=[[60.2259921875,137.65084375,1.51807287597656],[3.80360857770028E-05,0.00767312788400758,0.0049568441043783,-0.999958274808633],[0,0,0,0],[8.999999E+09,8.999999E+09,8.999999E+09,8.999999E+09,8.999999E+09,8.999999E+09]];
	LOCAL CONST Robtarget Tr_meulage_motif_2_P99 :=[[61.22390625,137.715421875,1.51772131347656],[3.80360857770028E-05,0.00767312788400758,0.0049568441043783,-0.999958274808633],[0,0,0,0],[8.999999E+09,8.999999E+09,8.999999E+09,8.999999E+09,8.999999E+09,8.999999E+09]];
	LOCAL CONST Robtarget Tr_meulage_motif_2_P100 :=[[62.2218203125,137.78,1.51736987304687],[3.80360857770028E-05,0.00767312788400758,0.0049568441043783,-0.999958274808633],[0,0,0,0],[8.999999E+09,8.999999E+09,8.999999E+09,8.999999E+09,8.999999E+09,8.999999E+09]];
	LOCAL CONST Robtarget Tr_meulage_motif_2_P101 :=[[63.21973046875,137.844578125,1.51701831054688],[3.80360857770028E-05,0.00767312788400758,0.0049568441043783,-0.999958274808633],[0,0,0,0],[8.999999E+09,8.999999E+09,8.999999E+09,8.999999E+09,8.999999E+09,8.999999E+09]];
	LOCAL CONST Robtarget Tr_meulage_motif_2_P102 :=[[64.21764453125,137.909140625,1.51666674804687],[3.80360857770028E-05,0.00767312788400758,0.0049568441043783,-0.999958274808633],[0,0,0,0],[8.999999E+09,8.999999E+09,8.999999E+09,8.999999E+09,8.999999E+09,8.999999E+09]];
	LOCAL CONST Robtarget Tr_meulage_motif_2_P103 :=[[65.2155546875,137.97371875,1.51631518554688],[3.80360857770028E-05,0.00767312788400758,0.0049568441043783,-0.999958274808633],[0,0,0,0],[8.999999E+09,8.999999E+09,8.999999E+09,8.999999E+09,8.999999E+09,8.999999E+09]];
	LOCAL CONST Robtarget Tr_meulage_motif_2_P104 :=[[66.21346875,138.038296875,1.51596362304687],[3.80360857770028E-05,0.00767312788400758,0.0049568441043783,-0.999958274808633],[0,0,0,0],[8.999999E+09,8.999999E+09,8.999999E+09,8.999999E+09,8.999999E+09,8.999999E+09]];
	LOCAL CONST Robtarget Tr_meulage_motif_2_P105 :=[[67.2113828125,138.102875,1.51561206054688],[3.80360857770028E-05,0.00767312788400758,0.0049568441043783,-0.999958274808633],[0,0,0,0],[8.999999E+09,8.999999E+09,8.999999E+09,8.999999E+09,8.999999E+09,8.999999E+09]];
	LOCAL CONST Robtarget Tr_meulage_motif_2_P106 :=[[68.209296875,138.167453125,1.51526049804688],[3.80360857770028E-05,0.00767312788400758,0.0049568441043783,-0.999958274808633],[0,0,0,0],[8.999999E+09,8.999999E+09,8.999999E+09,8.999999E+09,8.999999E+09,8.999999E+09]];
	LOCAL CONST Robtarget Tr_meulage_motif_2_P107 :=[[69.2072109375,138.23203125,1.51490893554688],[3.80360857770028E-05,0.00767312788400758,0.0049568441043783,-0.999958274808633],[0,0,0,0],[8.999999E+09,8.999999E+09,8.999999E+09,8.999999E+09,8.999999E+09,8.999999E+09]];
	LOCAL CONST Robtarget Tr_meulage_motif_2_P108 :=[[70.2051171875,138.296609375,1.51455749511719],[3.80360857770028E-05,0.00767312788400758,0.0049568441043783,-0.999958274808633],[0,0,0,0],[8.999999E+09,8.999999E+09,8.999999E+09,8.999999E+09,8.999999E+09,8.999999E+09]];
	LOCAL CONST Robtarget Tr_meulage_motif_2_P109 :=[[71.20303125,138.3611875,1.51420593261719],[3.80360857770028E-05,0.00767312788400758,0.0049568441043783,-0.999958274808633],[0,0,0,0],[8.999999E+09,8.999999E+09,8.999999E+09,8.999999E+09,8.999999E+09,8.999999E+09]];
	LOCAL CONST Robtarget Tr_meulage_motif_2_P110 :=[[72.2009453125,138.425765625,1.51385437011719],[3.80360857770028E-05,0.00767312788400758,0.0049568441043783,-0.999958274808633],[0,0,0,0],[8.999999E+09,8.999999E+09,8.999999E+09,8.999999E+09,8.999999E+09,8.999999E+09]];
	LOCAL CONST Robtarget Tr_meulage_motif_2_P111 :=[[73.198859375,138.49034375,1.51350280761719],[3.80360857770028E-05,0.00767312788400758,0.0049568441043783,-0.999958274808633],[0,0,0,0],[8.999999E+09,8.999999E+09,8.999999E+09,8.999999E+09,8.999999E+09,8.999999E+09]];
	LOCAL CONST Robtarget Tr_meulage_motif_2_P112 :=[[74.1967734375,138.55490625,1.51315124511719],[3.80360857770028E-05,0.00767312788400758,0.0049568441043783,-0.999958274808633],[0,0,0,0],[8.999999E+09,8.999999E+09,8.999999E+09,8.999999E+09,8.999999E+09,8.999999E+09]];
	LOCAL CONST Robtarget Tr_meulage_motif_2_P113 :=[[75.1946796875,138.619484375,1.51279968261719],[3.80360857770028E-05,0.00767312788400758,0.0049568441043783,-0.999958274808633],[0,0,0,0],[8.999999E+09,8.999999E+09,8.999999E+09,8.999999E+09,8.999999E+09,8.999999E+09]];
	LOCAL CONST Robtarget Tr_meulage_motif_2_P114 :=[[76.19259375,138.6840625,1.51244812011719],[3.80360857770028E-05,0.00767312788400758,0.0049568441043783,-0.999958274808633],[0,0,0,0],[8.999999E+09,8.999999E+09,8.999999E+09,8.999999E+09,8.999999E+09,8.999999E+09]];
	LOCAL CONST Robtarget Tr_meulage_motif_2_P115 :=[[77.1905078125,138.748640625,1.51209655761719],[3.80360857770028E-05,0.00767312788400758,0.0049568441043783,-0.999958274808633],[0,0,0,0],[8.999999E+09,8.999999E+09,8.999999E+09,8.999999E+09,8.999999E+09,8.999999E+09]];
	LOCAL CONST Robtarget Tr_meulage_motif_2_degg1 :=[[77.3439601961466,138.847779207697,-8.48623449848282],[3.80360857770028E-05,0.00767312788400758,0.0049568441043783,-0.999958274808633],[0,0,0,0],[8.999999E+09,8.999999E+09,8.999999E+09,8.999999E+09,8.999999E+09,8.999999E+09]];
	LOCAL CONST Robtarget Tr_meulage_motif_2_degg2 :=[[80.2595554854323,140.731412278944,-198.454524564383],[3.80360857770028E-05,0.00767312788400758,0.0049568441043783,-0.999958274808633],[0,0,0,0],[8.999999E+09,8.999999E+09,8.999999E+09,8.999999E+09,8.999999E+09,8.999999E+09]];
	LOCAL CONST Robtarget Tr_meulage_bavure_App1 :=[[-152.681627211269,280.571385972893,25.21126923728],[0.177388501312275,-0.179360733105625,0.68801010204285,-0.680444815182675],[0,0,0,0],[8.999999E+09,8.999999E+09,8.999999E+09,8.999999E+09,8.999999E+09,8.999999E+09]];
	LOCAL CONST Robtarget Tr_meulage_bavure_App2 :=[[-59.9273657355635,114.76356343927,23.110563461864],[0.177388501312275,-0.179360733105625,0.68801010204285,-0.680444815182675],[0,0,0,0],[8.999999E+09,8.999999E+09,8.999999E+09,8.999999E+09,8.999999E+09,8.999999E+09]];
	LOCAL CONST Robtarget Tr_meulage_bavure_P0 :=[[-55.0455625,106.0368359375,23],[0.177388501312275,-0.179360733105625,0.68801010204285,-0.680444815182675],[0,0,0,0],[8.999999E+09,8.999999E+09,8.999999E+09,8.999999E+09,8.999999E+09,8.999999E+09]];
	LOCAL CONST Robtarget Tr_meulage_bavure_P1 :=[[-58.557953125,103.9390546875,23],[0.177226846692387,-0.17919787394528,0.688053739755997,-0.68048572210793],[0,0,0,0],[8.999999E+09,8.999999E+09,8.999999E+09,8.999999E+09,8.999999E+09,8.999999E+09]];
	LOCAL CONST Robtarget Tr_meulage_bavure_P2 :=[[-61.01052734375,102.4794296875,23],[0.176749578650493,-0.17871609184946,0.688180649342477,-0.680608212433185],[0,0,0,0],[8.999999E+09,8.999999E+09,8.999999E+09,8.999999E+09,8.999999E+09,8.999999E+09]];
	LOCAL CONST Robtarget Tr_meulage_bavure_P3 :=[[-62.1965625,101.8155859375,23],[0.175976391053591,-0.177935383498329,0.688385129264931,-0.680806303509273],[0,0,0,0],[8.999999E+09,8.999999E+09,8.999999E+09,8.999999E+09,8.999999E+09,8.999999E+09]];
	LOCAL CONST Robtarget Tr_meulage_bavure_P4 :=[[-67.518765625,98.933046875,23],[0.174940822095379,-0.176889965879422,0.688657950951259,-0.681069655268375],[0,0,0,0],[8.999999E+09,8.999999E+09,8.999999E+09,8.999999E+09,8.999999E+09,8.999999E+09]];
	LOCAL CONST Robtarget Tr_meulage_bavure_P5 :=[[-68.2731640625,98.5295703125,23],[0.173686221300458,-0.175623974367364,0.688987241826052,-0.681385277767805],[0,0,0,0],[8.999999E+09,8.999999E+09,8.999999E+09,8.999999E+09,8.999999E+09,8.999999E+09]];
	LOCAL CONST Robtarget Tr_meulage_bavure_P6 :=[[-68.74615625,98.26821875,23],[0.172259853917705,-0.174183665358176,0.689356881467444,-0.681743121288453],[0,0,0,0],[8.999999E+09,8.999999E+09,8.999999E+09,8.999999E+09,8.999999E+09,8.999999E+09]];
	LOCAL CONST Robtarget Tr_meulage_bavure_P7 :=[[-70.4437265625,97.4023125,23],[0.170720749410025,-0.172629578642851,0.689752331177453,-0.682125484008433],[0,0,0,0],[8.999999E+09,8.999999E+09,8.999999E+09,8.999999E+09,8.999999E+09,8.999999E+09]];
	LOCAL CONST Robtarget Tr_meulage_bavure_P8 :=[[-76.1474609375,94.44275,23],[0.169122798255248,-0.17101651854432,0.690159881524304,-0.682517521701571],[0,0,0,0],[8.999999E+09,8.999999E+09,8.999999E+09,8.999999E+09,8.999999E+09,8.999999E+09]];
	LOCAL CONST Robtarget Tr_meulage_bavure_P9 :=[[-78.263765625,93.357359375,23],[0.167520768149853,-0.169399699896389,0.690565239121288,-0.682905692193918],[0,0,0,0],[8.999999E+09,8.999999E+09,8.999999E+09,8.999999E+09,8.999999E+09,8.999999E+09]];
	LOCAL CONST Robtarget Tr_meulage_bavure_P10 :=[[-78.6284453125,93.17334375,23],[0.165963476402512,-0.167828135819761,0.690955744246371,-0.683278860217847],[0,0,0,0],[8.999999E+09,8.999999E+09,8.999999E+09,8.999999E+09,8.999999E+09,8.999999E+09]];
	LOCAL CONST Robtarget Tr_meulage_bavure_P11 :=[[-78.997890625,92.9904453125,23],[0.164494861918919,-0.16634601937557,0.691320574818474,-0.683627314457836],[0,0,0,0],[8.999999E+09,8.999999E+09,8.999999E+09,8.999999E+09,8.999999E+09,8.999999E+09]];
	LOCAL CONST Robtarget Tr_meulage_bavure_P12 :=[[-83.8377109375,90.681703125,23],[0.163150367663531,-0.164989804019774,0.691652969713093,-0.68394187734619],[0,0,0,0],[8.999999E+09,8.999999E+09,8.999999E+09,8.999999E+09,8.999999E+09,8.999999E+09]];
	LOCAL CONST Robtarget Tr_meulage_bavure_P13 :=[[-87.449765625,88.955171875,23],[0.161952533026557,-0.163781934608315,0.691947640045025,-0.684218765000171],[0,0,0,0],[8.999999E+09,8.999999E+09,8.999999E+09,8.999999E+09,8.999999E+09,8.999999E+09]];
	LOCAL CONST Robtarget Tr_meulage_bavure_P14 :=[[-89.1013203125,88.20325,23],[0.160917799905264,-0.162739226848267,0.692201857201547,-0.684454523401816],[0,0,0,0],[8.999999E+09,8.999999E+09,8.999999E+09,8.999999E+09,8.999999E+09,8.999999E+09]];
	LOCAL CONST Robtarget Tr_meulage_bavure_P15 :=[[-93.006015625,86.2990390625,23],[0.16004830555267,-0.161863422438848,0.692415054654168,-0.684650395789243],[0,0,0,0],[8.999999E+09,8.999999E+09,8.999999E+09,8.999999E+09,8.999999E+09,8.999999E+09]];
	LOCAL CONST Robtarget Tr_meulage_bavure_P16 :=[[-93.31903125,86.1553359375,23],[0.159340683605488,-0.161150589467166,0.692587606994267,-0.684809054189907],[0,0,0,0],[8.999999E+09,8.999999E+09,8.999999E+09,8.999999E+09,8.999999E+09,8.999999E+09]];
	LOCAL CONST Robtarget Tr_meulage_bavure_P17 :=[[-94.1096796875,85.7535078125,23],[0.158779926018583,-0.160586846791741,0.692726141303789,-0.68493159723098],[0,0,0,0],[8.999999E+09,8.999999E+09,8.999999E+09,8.999999E+09,8.999999E+09,8.999999E+09]];
	LOCAL CONST Robtarget Tr_meulage_bavure_P18 :=[[-97.9572734375,83.8231171875,23],[0.158347170839766,-0.160152143577062,0.692833475996657,-0.68502499146608],[0,0,0,0],[8.999999E+09,8.999999E+09,8.999999E+09,8.999999E+09,8.999999E+09,8.999999E+09]];
	LOCAL CONST Robtarget Tr_meulage_bavure_P19 :=[[-101.1501796875,82.188296875,23],[0.158019746982021,-0.159823311550329,0.692914650976008,-0.68509528907417],[0,0,0,0],[8.999999E+09,8.999999E+09,8.999999E+09,8.999999E+09,8.999999E+09,8.999999E+09]];
	LOCAL CONST Robtarget Tr_meulage_bavure_P20 :=[[-101.6714765625,81.9326484375,23],[0.157771932232446,-0.159575772726041,0.692978717561331,-0.685145303687896],[0,0,0,0],[8.999999E+09,8.999999E+09,8.999999E+09,8.999999E+09,8.999999E+09,8.999999E+09]];
	LOCAL CONST Robtarget Tr_meulage_bavure_P21 :=[[-102.3454609375,81.602046875,23],[0.157580166884127,-0.159384424832202,0.693028658825587,-0.685183460229512],[0,0,0,0],[8.999999E+09,8.999999E+09,8.999999E+09,8.999999E+09,8.999999E+09,8.999999E+09]];
	LOCAL CONST Robtarget Tr_meulage_bavure_P22 :=[[-108.2710546875,78.7345,23],[0.157425756575583,-0.159229876201055,0.693067875449075,-0.685215219994498],[0,0,0,0],[8.999999E+09,8.999999E+09,8.999999E+09,8.999999E+09,8.999999E+09,8.999999E+09]];
	LOCAL CONST Robtarget Tr_meulage_bavure_P23 :=[[-111.588046875,77.1989765625,23],[0.157287671596977,-0.159091544370672,0.693102669943371,-0.685243867386441],[0,0,0,0],[8.999999E+09,8.999999E+09,8.999999E+09,8.999999E+09,8.999999E+09,8.999999E+09]];
	LOCAL CONST Robtarget Tr_meulage_bavure_P24 :=[[-115.1573203125,75.4651796875,23],[0.15715223428919,-0.1589555491293,0.693136129825429,-0.685272656823213],[0,0,0,0],[8.999999E+09,8.999999E+09,8.999999E+09,8.999999E+09,8.999999E+09,8.999999E+09]];
	LOCAL CONST Robtarget Tr_meulage_bavure_P25 :=[[-118.3474453125,73.936765625,23],[0.157008520359977,-0.158810273050823,0.693169627145671,-0.68530539886289],[0,0,0,0],[8.999999E+09,8.999999E+09,8.999999E+09,8.999999E+09,8.999999E+09,8.999999E+09]];
	LOCAL CONST Robtarget Tr_meulage_bavure_P26 :=[[-119.0849609375,73.5809296875,23],[0.156851431032105,-0.158651277473044,0.693205799611552,-0.685341608341608],[0,0,0,0],[8.999999E+09,8.999999E+09,8.999999E+09,8.999999E+09,8.999999E+09,8.999999E+09]];
	LOCAL CONST Robtarget Tr_meulage_bavure_P27 :=[[-125.9613984375,70.2841171875,23],[0.156675879121197,-0.158472539345323,0.693244016276487,-0.685384459316004],[0,0,0,0],[8.999999E+09,8.999999E+09,8.999999E+09,8.999999E+09,8.999999E+09,8.999999E+09]];
	LOCAL CONST Robtarget Tr_meulage_bavure_P28 :=[[-130.8094140625,67.94915625,23],[0.156478837924113,-0.158271132212213,0.693285227787676,-0.685434325753805],[0,0,0,0],[8.999999E+09,8.999999E+09,8.999999E+09,8.999999E+09,8.999999E+09,8.999999E+09]];
	LOCAL CONST Robtarget Tr_meulage_bavure_P29 :=[[-132.24225,67.28134375,23],[0.156262841141247,-0.158049965687939,0.693329531879704,-0.685489819798936],[0,0,0,0],[8.999999E+09,8.999999E+09,8.999999E+09,8.999999E+09,8.999999E+09,8.999999E+09]];
	LOCAL CONST Robtarget Tr_meulage_bavure_P30 :=[[-137.107453125,64.9970703125,23],[0.15602864718163,-0.15780930372763,0.693375691720953,-0.685551920022227],[0,0,0,0],[8.999999E+09,8.999999E+09,8.999999E+09,8.999999E+09,8.999999E+09,8.999999E+09]];
	LOCAL CONST Robtarget Tr_meulage_bavure_P31 :=[[-142.82559375,62.2412421875,23],[0.155781290059968,-0.157554268048919,0.693422577993565,-0.685619406533668],[0,0,0,0],[8.999999E+09,8.999999E+09,8.999999E+09,8.999999E+09,8.999999E+09,8.999999E+09]];
	LOCAL CONST Robtarget Tr_meulage_bavure_P32 :=[[-143.9945,61.66491796875,23],[0.155524705604104,-0.157287615008368,0.693466729431039,-0.685694222874857],[0,0,0,0],[8.999999E+09,8.999999E+09,8.999999E+09,8.999999E+09,8.999999E+09,8.999999E+09]];
	LOCAL CONST Robtarget Tr_meulage_bavure_P33 :=[[-145.9565625,60.74685546875,23],[0.155266299181018,-0.15701891771228,0.693510720421759,-0.685769871370263],[0,0,0,0],[8.999999E+09,8.999999E+09,8.999999E+09,8.999999E+09,8.999999E+09,8.999999E+09]];
	LOCAL CONST Robtarget Tr_meulage_bavure_P34 :=[[-147.61965625,59.9593828125,23],[0.155013264246003,-0.156753607421948,0.693549080216587,-0.685849012391745],[0,0,0,0],[8.999999E+09,8.999999E+09,8.999999E+09,8.999999E+09,8.999999E+09,8.999999E+09]];
	LOCAL CONST Robtarget Tr_meulage_bavure_P35 :=[[-150.451859375,58.62628125,23],[0.1547721827214,-0.156498898436797,0.693581451149887,-0.685928886156968],[0,0,0,0],[8.999999E+09,8.999999E+09,8.999999E+09,8.999999E+09,8.999999E+09,8.999999E+09]];
	LOCAL CONST Robtarget Tr_meulage_bavure_P36 :=[[-157.15275,55.47647265625,23],[0.154552162941699,-0.156264571077962,0.693606948246835,-0.686006132698226],[0,0,0,0],[8.999999E+09,8.999999E+09,8.999999E+09,8.999999E+09,8.999999E+09,8.999999E+09]];
	LOCAL CONST Robtarget Tr_meulage_bavure_P37 :=[[-161.192953125,53.51309375,23],[0.15435774579128,-0.156053989879853,0.693622005392172,-0.686082613241697],[0,0,0,0],[8.999999E+09,8.999999E+09,8.999999E+09,8.999999E+09,8.999999E+09,8.999999E+09]];
	LOCAL CONST Robtarget Tr_meulage_bavure_P38 :=[[-165.307296875,51.5829765625,23],[0.154191979416759,-0.155870496939621,0.693626492560407,-0.686157059634079],[0,0,0,0],[8.999999E+09,8.999999E+09,8.999999E+09,8.999999E+09,8.999999E+09,8.999999E+09]];
	LOCAL CONST Robtarget Tr_meulage_bavure_P39 :=[[-165.44575,51.522125,23],[0.154057715801509,-0.155717983728721,0.693621897368158,-0.686226488294411],[0,0,0,0],[8.999999E+09,8.999999E+09,8.999999E+09,8.999999E+09,8.999999E+09,8.999999E+09]];
	LOCAL CONST Robtarget Tr_meulage_bavure_P40 :=[[-165.530921875,51.48303125,23],[0.153955291355828,-0.155595404269901,0.693605282233213,-0.68629407027295],[0,0,0,0],[8.999999E+09,8.999999E+09,8.999999E+09,8.999999E+09,8.999999E+09,8.999999E+09]];
	LOCAL CONST Robtarget Tr_meulage_bavure_P41 :=[[-165.871640625,51.319609375,23],[0.153881487266343,-0.155499479756811,0.693577351569644,-0.686360588219995],[0,0,0,0],[8.999999E+09,8.999999E+09,8.999999E+09,8.999999E+09,8.999999E+09,8.999999E+09]];
	LOCAL CONST Robtarget Tr_meulage_bavure_P42 :=[[-170.717265625,49.040375,23],[0.15383055741581,-0.15542527646801,0.693541260495935,-0.686425278547996],[0,0,0,0],[8.999999E+09,8.999999E+09,8.999999E+09,8.999999E+09,8.999999E+09,8.999999E+09]];
	LOCAL CONST Robtarget Tr_meulage_bavure_P43 :=[[-172.865828125,47.9996953125,23],[0.153806187374644,-0.155374736497753,0.693492466424944,-0.686491476272924],[0,0,0,0],[8.999999E+09,8.999999E+09,8.999999E+09,8.999999E+09,8.999999E+09,8.999999E+09]];
	LOCAL CONST Robtarget Tr_meulage_bavure_P44 :=[[-175.658984375,46.73690625,23],[0.153804253723473,-0.155344969042178,0.693434599498108,-0.686557097661039],[0,0,0,0],[8.999999E+09,8.999999E+09,8.999999E+09,8.999999E+09,8.999999E+09,8.999999E+09]];
	LOCAL CONST Robtarget Tr_meulage_bavure_P45 :=[[-178.551015625,45.4736328125,23],[0.153828245397285,-0.155338719504123,0.693365265520501,-0.686623158443187],[0,0,0,0],[8.999999E+09,8.999999E+09,8.999999E+09,8.999999E+09,8.999999E+09,8.999999E+09]];
	LOCAL CONST Robtarget Tr_meulage_bavure_P46 :=[[-179.940359375,44.8505546875,23],[0.153885425822735,-0.155363972537814,0.693284219274807,-0.686686466344828],[0,0,0,0],[8.999999E+09,8.999999E+09,8.999999E+09,8.999999E+09,8.999999E+09,8.999999E+09]];
	LOCAL CONST Robtarget Tr_meulage_bavure_P47 :=[[-181.251390625,44.222625,23],[0.153984506790743,-0.155428367174819,0.693187112731023,-0.686747712838862],[0,0,0,0],[8.999999E+09,8.999999E+09,8.999999E+09,8.999999E+09,8.999999E+09,8.999999E+09]];
	LOCAL CONST Robtarget Tr_meulage_bavure_P48 :=[[-184.561578125,42.6696796875,23],[0.154138861700727,-0.155545634707039,0.693071469962167,-0.686803250110007],[0,0,0,0],[8.999999E+09,8.999999E+09,8.999999E+09,8.999999E+09,8.999999E+09,8.999999E+09]];
	LOCAL CONST Robtarget Tr_meulage_bavure_P49 :=[[-187.78425,41.11605859375,23],[0.15436154152056,-0.15572887245607,0.692934261997497,-0.686850159301825],[0,0,0,0],[8.999999E+09,8.999999E+09,8.999999E+09,8.999999E+09,8.999999E+09,8.999999E+09]];
	LOCAL CONST Robtarget Tr_meulage_bavure_P50 :=[[-189.367015625,40.33508203125,23],[0.154669867206225,-0.155995404377384,0.692771337345859,-0.686884662911886],[0,0,0,0],[8.999999E+09,8.999999E+09,8.999999E+09,8.999999E+09,8.999999E+09,8.999999E+09]];
	LOCAL CONST Robtarget Tr_meulage_bavure_P51 :=[[-192.489296875,38.87896875,23],[0.155064948483069,-0.156345784355804,0.692581358012916,-0.686907504689748],[0,0,0,0],[8.999999E+09,8.999999E+09,8.999999E+09,8.999999E+09,8.999999E+09,8.999999E+09]];
	LOCAL CONST Robtarget Tr_meulage_bavure_P52 :=[[-196.19278125,37.2769765625,23],[0.155558739194606,-0.156793107743898,0.692363858487139,-0.686913158619775],[0,0,0,0],[8.999999E+09,8.999999E+09,8.999999E+09,8.999999E+09,8.999999E+09,8.999999E+09]];
	LOCAL CONST Robtarget Tr_meulage_bavure_P53 :=[[-200.52359375,35.36804296875,23],[0.156157533353722,-0.157341901589033,0.692113695863833,-0.686903910877594],[0,0,0,0],[8.999999E+09,8.999999E+09,8.999999E+09,8.999999E+09,8.999999E+09,8.999999E+09]];
	LOCAL CONST Robtarget Tr_meulage_bavure_P54 :=[[-206.424828125,32.55514453125,23],[0.156858249651062,-0.157989965371902,0.69183350941289,-0.686877758856432],[0,0,0,0],[8.999999E+09,8.999999E+09,8.999999E+09,8.999999E+09,8.999999E+09,8.999999E+09]];
	LOCAL CONST Robtarget Tr_meulage_bavure_P55 :=[[-207.687890625,31.94403125,23],[0.157666698227001,-0.158742956141727,0.691521586372181,-0.686833154213514],[0,0,0,0],[8.999999E+09,8.999999E+09,8.999999E+09,8.999999E+09,8.999999E+09,8.999999E+09]];
	LOCAL CONST Robtarget Tr_meulage_bavure_P56 :=[[-210.21653125,30.681609375,23],[0.158582241567178,-0.15960002098923,0.691177641008899,-0.686769957503341],[0,0,0,0],[8.999999E+09,8.999999E+09,8.999999E+09,8.999999E+09,8.999999E+09,8.999999E+09]];
	LOCAL CONST Robtarget Tr_meulage_bavure_P57 :=[[-212.55865625,29.466125,23],[0.159629065846824,-0.160584415911483,0.69079381684606,-0.68668414086135],[0,0,0,0],[8.999999E+09,8.999999E+09,8.999999E+09,8.999999E+09,8.999999E+09,8.999999E+09]];
	LOCAL CONST Robtarget Tr_meulage_bavure_P58 :=[[-213.65040625,28.86767578125,23],[0.160837467857986,-0.161726139253885,0.690361978829387,-0.686568498404812],[0,0,0,0],[8.999999E+09,8.999999E+09,8.999999E+09,8.999999E+09,8.999999E+09,8.999999E+09]];
	LOCAL CONST Robtarget Tr_meulage_bavure_P59 :=[[-218.437578125,26.28790234375,23],[0.162264622863535,-0.163082780146969,0.689868617838609,-0.686407669761882],[0,0,0,0],[8.999999E+09,8.999999E+09,8.999999E+09,8.999999E+09,8.999999E+09,8.999999E+09]];
	LOCAL CONST Robtarget Tr_meulage_bavure_P60 :=[[-219.236265625,25.872345703125,23],[0.163975257482769,-0.164718181745359,0.68929539646674,-0.686186484817154],[0,0,0,0],[8.999999E+09,8.999999E+09,8.999999E+09,8.999999E+09,8.999999E+09,8.999999E+09]];
	LOCAL CONST Robtarget Tr_meulage_bavure_P61 :=[[-225.322515625,22.81921484375,23],[0.166076202997506,-0.166740079046899,0.688616337572651,-0.685874609870779],[0,0,0,0],[8.999999E+09,8.999999E+09,8.999999E+09,8.999999E+09,8.999999E+09,8.999999E+09]];
	LOCAL CONST Robtarget Tr_meulage_bavure_P62 :=[[-227.205625,21.884705078125,23],[0.168710262911837,-0.169290893528402,0.687792428340487,-0.685433451236566],[0,0,0,0],[8.999999E+09,8.999999E+09,8.999999E+09,8.999999E+09,8.999999E+09,8.999999E+09]];
	LOCAL CONST Robtarget Tr_meulage_bavure_P63 :=[[-227.81334375,21.592345703125,23],[0.172027810134917,-0.172519679367679,0.686778375964267,-0.684820308605799],[0,0,0,0],[8.999999E+09,8.999999E+09,8.999999E+09,8.999999E+09,8.999999E+09,8.999999E+09]];
	LOCAL CONST Robtarget Tr_meulage_bavure_P64 :=[[-229.4960625,20.7865,23],[0.176212910849779,-0.176610394290867,0.685518305024735,-0.683975461660934],[0,0,0,0],[8.999999E+09,8.999999E+09,8.999999E+09,8.999999E+09,8.999999E+09,8.999999E+09]];
	LOCAL CONST Robtarget Tr_meulage_bavure_P65 :=[[-233.728171875,18.802826171875,23],[0.181459699502922,-0.181754396747503,0.683942028486953,-0.682833082376954],[0,0,0,0],[8.999999E+09,8.999999E+09,8.999999E+09,8.999999E+09,8.999999E+09,8.999999E+09]];
	LOCAL CONST Robtarget Tr_meulage_bavure_P66 :=[[-237.41315625,16.984587890625,23],[0.187974550703908,-0.188157720151535,0.681970419963907,-0.681306529345854],[0,0,0,0],[8.999999E+09,8.999999E+09,8.999999E+09,8.999999E+09,8.999999E+09,8.999999E+09]];
	LOCAL CONST Robtarget Tr_meulage_bavure_P67 :=[[-238.5531875,16.454345703125,23],[0.195980659243853,-0.19603841902724,0.679497076871882,-0.679296873237477],[0,0,0,0],[8.999999E+09,8.999999E+09,8.999999E+09,8.999999E+09,8.999999E+09,8.999999E+09]];
	LOCAL CONST Robtarget Tr_meulage_bavure_P68 :=[[-239.62603125,15.86346484375,23],[0.205689154807885,-0.205604941392757,0.676403618985205,-0.676680666114392],[0,0,0,0],[8.999999E+09,8.999999E+09,8.999999E+09,8.999999E+09,8.999999E+09,8.999999E+09]];
	LOCAL CONST Robtarget Tr_meulage_bavure_P69 :=[[-241.881015625,14.674072265625,23],[0.217315068469975,-0.217067684449807,0.672541532954208,-0.673308003691545],[0,0,0,0],[8.999999E+09,8.999999E+09,8.999999E+09,8.999999E+09,8.999999E+09,8.999999E+09]];
	LOCAL CONST Robtarget Tr_meulage_bavure_P70 :=[[-243.19428125,13.981994140625,23],[0.231043030485618,-0.230605026616671,0.667736878916933,-0.669005157153082],[0,0,0,0],[8.999999E+09,8.999999E+09,8.999999E+09,8.999999E+09,8.999999E+09,8.999999E+09]];
	LOCAL CONST Robtarget Tr_meulage_bavure_P71 :=[[-244.81090625,13.240142578125,23],[0.247079601554136,-0.246419216261593,0.661769901321302,-0.663543395761021],[0,0,0,0],[8.999999E+09,8.999999E+09,8.999999E+09,8.999999E+09,8.999999E+09,8.999999E+09]];
	LOCAL CONST Robtarget Tr_meulage_bavure_P72 :=[[-245.96340625,12.702208984375,23],[0.265606175583457,-0.264683539413277,0.654372032820531,-0.656653048510335],[0,0,0,0],[8.999999E+09,8.999999E+09,8.999999E+09,8.999999E+09,8.999999E+09,8.999999E+09]];
	LOCAL CONST Robtarget Tr_meulage_bavure_P73 :=[[-247.046859375,11.9559326171875,23],[0.286765810247674,-0.28553143232641,0.645224711758096,-0.648014075899055],[0,0,0,0],[8.999999E+09,8.999999E+09,8.999999E+09,8.999999E+09,8.999999E+09,8.999999E+09]];
	LOCAL CONST Robtarget Tr_meulage_bavure_P74 :=[[-248.908984375,10.6868896484375,23],[0.310627630821205,-0.309026362897003,0.63397049769814,-0.637255513945095],[0,0,0,0],[8.999999E+09,8.999999E+09,8.999999E+09,8.999999E+09,8.999999E+09,8.999999E+09]];
	LOCAL CONST Robtarget Tr_meulage_bavure_P75 :=[[-249.20990625,10.5189208984375,23],[0.337164197846283,-0.33513356223183,0.620213739106412,-0.623971727708972],[0,0,0,0],[8.999999E+09,8.999999E+09,8.999999E+09,8.999999E+09,8.999999E+09,8.999999E+09]];
	LOCAL CONST Robtarget Tr_meulage_bavure_P76 :=[[-250.342453125,9.464263671875,23],[0.366208120872859,-0.363671905981819,0.603546144634793,-0.607755220712088],[0,0,0,0],[8.999999E+09,8.999999E+09,8.999999E+09,8.999999E+09,8.999999E+09,8.999999E+09]];
	LOCAL CONST Robtarget Tr_meulage_bavure_P77 :=[[-250.983765625,8.8249814453125,23],[0.397290392191781,-0.394175843200127,0.583686818539605,-0.588298773390429],[0,0,0,0],[8.999999E+09,8.999999E+09,8.999999E+09,8.999999E+09,8.999999E+09,8.999999E+09]];
	LOCAL CONST Robtarget Tr_meulage_bavure_P78 :=[[-251.919109375,5.6274716796875,23],[0.429653654209421,-0.425883437787876,0.560550213119632,-0.565512593506109],[0,0,0,0],[8.999999E+09,8.999999E+09,8.999999E+09,8.999999E+09,8.999999E+09,8.999999E+09]];
	LOCAL CONST Robtarget Tr_meulage_bavure_P79 :=[[-252.046296875,5.2871396484375,23],[0.462217707676489,-0.457718708503253,0.534418512366918,-0.53967140765093],[0,0,0,0],[8.999999E+09,8.999999E+09,8.999999E+09,8.999999E+09,8.999999E+09,8.999999E+09]];
	LOCAL CONST Robtarget Tr_meulage_bavure_P80 :=[[-252.067890625,5.1832578125,23],[0.493767019384114,-0.488476554177658,0.505969079208182,-0.511448997919122],[0,0,0,0],[8.999999E+09,8.999999E+09,8.999999E+09,8.999999E+09,8.999999E+09,8.999999E+09]];
	LOCAL CONST Robtarget Tr_meulage_bavure_P81 :=[[-251.8983125,4.776611328125,23],[0.523084177234694,-0.516954864759415,0.476302975038361,-0.481950295464049],[0,0,0,0],[8.999999E+09,8.999999E+09,8.999999E+09,8.999999E+09,8.999999E+09,8.999999E+09]];
	LOCAL CONST Robtarget Tr_meulage_bavure_P82 :=[[-251.0103125,2.58804321289063,23],[0.549265657191203,-0.542272338201529,0.446692428088128,-0.452453117726572],[0,0,0,0],[8.999999E+09,8.999999E+09,8.999999E+09,8.999999E+09,8.999999E+09,8.999999E+09]];
	LOCAL CONST Robtarget Tr_meulage_bavure_P83 :=[[-249.440296875,0.626129150390625,23],[0.571796085303502,-0.563925507393734,0.418399726215847,-0.424239234447753],[0,0,0,0],[8.999999E+09,8.999999E+09,8.999999E+09,8.999999E+09,8.999999E+09,8.999999E+09]];
	LOCAL CONST Robtarget Tr_meulage_bavure_P84 :=[[-248.982390625,0.053955078125,23],[0.59060922516294,-0.581859544440979,0.39239937956523,-0.398300063535259],[0,0,0,0],[8.999999E+09,8.999999E+09,8.999999E+09,8.999999E+09,8.999999E+09,8.999999E+09]];
	LOCAL CONST Robtarget Tr_meulage_bavure_P85 :=[[-248.341109375,-0.583404541015625,23],[0.605930333124081,-0.596307475253473,0.369342369488412,-0.375302598522384],[0,0,0,0],[8.999999E+09,8.999999E+09,8.999999E+09,8.999999E+09,8.999999E+09,8.999999E+09]];
	LOCAL CONST Robtarget Tr_meulage_bavure_P86 :=[[-246.566390625,-2.4132080078125,23],[0.618198415561435,-0.607717002833619,0.349472178115758,-0.355499592386942],[0,0,0,0],[8.999999E+09,8.999999E+09,8.999999E+09,8.999999E+09,8.999999E+09,8.999999E+09]];
	LOCAL CONST Robtarget Tr_meulage_bavure_P87 :=[[-245.520125,-3.32345581054688,23],[0.62788394884294,-0.616554075067624,0.332802369724062,-0.338917987142836],[0,0,0,0],[8.999999E+09,8.999999E+09,8.999999E+09,8.999999E+09,8.999999E+09,8.999999E+09]];
	LOCAL CONST Robtarget Tr_meulage_bavure_P88 :=[[-243.9953125,-4.7114560546875,23],[0.635446404937751,-0.623277730763268,0.319152481844011,-0.325383512365159],[0,0,0,0],[8.999999E+09,8.999999E+09,8.999999E+09,8.999999E+09,8.999999E+09,8.999999E+09]];
	LOCAL CONST Robtarget Tr_meulage_bavure_P89 :=[[-235.859125,-12.962890625,23],[0.641290784795364,-0.628294535237666,0.308237635163517,-0.314613519410456],[0,0,0,0],[8.999999E+09,8.999999E+09,8.999999E+09,8.999999E+09,8.999999E+09,8.999999E+09]];
	LOCAL CONST Robtarget Tr_meulage_bavure_P90 :=[[-234.935984375,-13.9076845703125,23],[0.645776076312793,-0.631965450548974,0.299687019134427,-0.306236214606972],[0,0,0,0],[8.999999E+09,8.999999E+09,8.999999E+09,8.999999E+09,8.999999E+09,8.999999E+09]];
	LOCAL CONST Robtarget Tr_meulage_bavure_P91 :=[[-234.783546875,-14.0496826171875,23],[0.649195189814487,-0.634582562062778,0.293127830580057,-0.299877729061366],[0,0,0,0],[8.999999E+09,8.999999E+09,8.999999E+09,8.999999E+09,8.999999E+09,8.999999E+09]];
	LOCAL CONST Robtarget Tr_meulage_bavure_P92 :=[[-234.254625,-14.6212158203125,23],[0.651782077550716,-0.63636990085114,0.28821953065408,-0.295199889606897],[0,0,0,0],[8.999999E+09,8.999999E+09,8.999999E+09,8.999999E+09,8.999999E+09,8.999999E+09]];
	LOCAL CONST Robtarget Tr_meulage_bavure_P93 :=[[-229.82184375,-19.5146796875,23],[0.653737578743892,-0.637535231016826,0.284610655648542,-0.29184376306802],[0,0,0,0],[8.999999E+09,8.999999E+09,8.999999E+09,8.999999E+09,8.999999E+09,8.999999E+09]];
	LOCAL CONST Robtarget Tr_meulage_bavure_P94 :=[[-227.59946875,-21.936919921875,23],[0.655220721649949,-0.638235380776988,0.282003747874267,-0.289508705965537],[0,0,0,0],[8.999999E+09,8.999999E+09,8.999999E+09,8.999999E+09,8.999999E+09,8.999999E+09]];
	LOCAL CONST Robtarget Tr_meulage_bavure_P95 :=[[-223.917796875,-25.985626953125,23],[0.656367083510457,-0.638599262238533,0.280130117839521,-0.287924210568673],[0,0,0,0],[8.999999E+09,8.999999E+09,8.999999E+09,8.999999E+09,8.999999E+09,8.999999E+09]];
	LOCAL CONST Robtarget Tr_meulage_bavure_P96 :=[[-219.656671875,-30.4964296875,23],[0.657277448443186,-0.63873196576186,0.278773605980662,-0.286867754009653],[0,0,0,0],[8.999999E+09,8.999999E+09,8.999999E+09,8.999999E+09,8.999999E+09,8.999999E+09]];
	LOCAL CONST Robtarget Tr_meulage_bavure_P97 :=[[-218.16828125,-32.04049609375,23],[0.658035384380299,-0.638714649889351,0.277754480358638,-0.286156386545712],[0,0,0,0],[8.999999E+09,8.999999E+09,8.999999E+09,8.999999E+09,8.999999E+09,8.999999E+09]];
	LOCAL CONST Robtarget Tr_meulage_bavure_P98 :=[[-216.249125,-34.02264453125,23],[0.658704192073494,-0.638614149034684,0.276929337171777,-0.285641205380303],[0,0,0,0],[8.999999E+09,8.999999E+09,8.999999E+09,8.999999E+09,8.999999E+09,8.999999E+09]];
	LOCAL CONST Robtarget Tr_meulage_bavure_P99 :=[[-214.91665625,-35.41192578125,23],[0.659329411147182,-0.638474901511729,0.276197171149646,-0.285218601049846],[0,0,0,0],[8.999999E+09,8.999999E+09,8.999999E+09,8.999999E+09,8.999999E+09,8.999999E+09]];
	LOCAL CONST Robtarget Tr_meulage_bavure_P100 :=[[-210.074421875,-40.50796484375,23],[0.659958336031171,-0.638336665675489,0.275457841866844,-0.284788120031941],[0,0,0,0],[8.999999E+09,8.999999E+09,8.999999E+09,8.999999E+09,8.999999E+09,8.999999E+09]];
	LOCAL CONST Robtarget Tr_meulage_bavure_P101 :=[[-207.8455625,-42.93337890625,23],[0.660621878048134,-0.638238210824234,0.274633912922375,-0.284265605307751],[0,0,0,0],[8.999999E+09,8.999999E+09,8.999999E+09,8.999999E+09,8.999999E+09,8.999999E+09]];
	LOCAL CONST Robtarget Tr_meulage_bavure_P102 :=[[-202.855828125,-48.38467578125,23],[0.661333336085144,-0.638189413465173,0.27369757766831,-0.283623213263603],[0,0,0,0],[8.999999E+09,8.999999E+09,8.999999E+09,8.999999E+09,8.999999E+09,8.999999E+09]];
	LOCAL CONST Robtarget Tr_meulage_bavure_P103 :=[[-198.896125,-52.569625,23],[0.662110738734719,-0.638209740246365,0.272605361779014,-0.282814451250576],[0,0,0,0],[8.999999E+09,8.999999E+09,8.999999E+09,8.999999E+09,8.999999E+09,8.999999E+09]];
	LOCAL CONST Robtarget Tr_meulage_bavure_P104 :=[[-198.54165625,-52.95010546875,23],[0.662963158629786,-0.638311750579175,0.271331645859519,-0.281810392511226],[0,0,0,0],[8.999999E+09,8.999999E+09,8.999999E+09,8.999999E+09,8.999999E+09,8.999999E+09]];
	LOCAL CONST Robtarget Tr_meulage_bavure_P105 :=[[-195.9013125,-55.72535546875,23],[0.663902040334473,-0.638500426218784,0.269853594644861,-0.280589244297429],[0,0,0,0],[8.999999E+09,8.999999E+09,8.999999E+09,8.999999E+09,8.999999E+09,8.999999E+09]];
	LOCAL CONST Robtarget Tr_meulage_bavure_P106 :=[[-193.729140625,-58.024078125,23],[0.664913756274626,-0.638770061442384,0.26819239700557,-0.279169023192164],[0,0,0,0],[8.999999E+09,8.999999E+09,8.999999E+09,8.999999E+09,8.999999E+09,8.999999E+09]];
	LOCAL CONST Robtarget Tr_meulage_bavure_P107 :=[[-193.28953125,-58.51324609375,23],[0.665995325925427,-0.639118284040195,0.26635109810518,-0.277552044469437],[0,0,0,0],[8.999999E+09,8.999999E+09,8.999999E+09,8.999999E+09,8.999999E+09,8.999999E+09]];
	LOCAL CONST Robtarget Tr_meulage_bavure_P108 :=[[-191.9241875,-59.996703125,23],[0.667131620849257,-0.639529335541131,0.264362177577655,-0.275772131499474],[0,0,0,0],[8.999999E+09,8.999999E+09,8.999999E+09,8.999999E+09,8.999999E+09,8.999999E+09]];
	LOCAL CONST Robtarget Tr_meulage_bavure_P109 :=[[-188.98003125,-63.22674609375,23],[0.668298485469852,-0.639979293863926,0.262279393008099,-0.273885300349316],[0,0,0,0],[8.999999E+09,8.999999E+09,8.999999E+09,8.999999E+09,8.999999E+09,8.999999E+09]];
	LOCAL CONST Robtarget Tr_meulage_bavure_P110 :=[[-185.510671875,-66.9500390625,23],[0.669471046156276,-0.640449996889709,0.260153536335568,-0.271942011051052],[0,0,0,0],[8.999999E+09,8.999999E+09,8.999999E+09,8.999999E+09,8.999999E+09,8.999999E+09]];
	LOCAL CONST Robtarget Tr_meulage_bavure_P111 :=[[-183.67946875,-68.9160625,23],[0.670619976730549,-0.640909623203705,0.258056709438292,-0.270019325991093],[0,0,0,0],[8.999999E+09,8.999999E+09,8.999999E+09,8.999999E+09,8.999999E+09,8.999999E+09]];
	LOCAL CONST Robtarget Tr_meulage_bavure_P112 :=[[-182.063140625,-70.4321015625,23],[0.671706698281797,-0.641323889787921,0.256079283112639,-0.268211074773532],[0,0,0,0],[8.999999E+09,8.999999E+09,8.999999E+09,8.999999E+09,8.999999E+09,8.999999E+09]];
	LOCAL CONST Robtarget Tr_meulage_bavure_P113 :=[[-180.931953125,-71.4937734375,23],[0.672698394866022,-0.641666617987956,0.254297845933301,-0.266595998578859],[0,0,0,0],[8.999999E+09,8.999999E+09,8.999999E+09,8.999999E+09,8.999999E+09,8.999999E+09]];
	LOCAL CONST Robtarget Tr_meulage_bavure_P114 :=[[-179.544515625,-72.66459375,23],[0.673567278126777,-0.641909053604419,0.252785915565448,-0.265253029444157],[0,0,0,0],[8.999999E+09,8.999999E+09,8.999999E+09,8.999999E+09,8.999999E+09,8.999999E+09]];
	LOCAL CONST Robtarget Tr_meulage_bavure_P115 :=[[-179.0376875,-73.0277265625,23],[0.67429016163862,-0.642031459858704,0.251602090342396,-0.264243771174274],[0,0,0,0],[8.999999E+09,8.999999E+09,8.999999E+09,8.999999E+09,8.999999E+09,8.999999E+09]];
	LOCAL CONST Robtarget Tr_meulage_bavure_P116 :=[[-176.7835625,-74.7749453125,23],[0.67484470408022,-0.642010705866188,0.250806908225722,-0.26363378712588],[0,0,0,0],[8.999999E+09,8.999999E+09,8.999999E+09,8.999999E+09,8.999999E+09,8.999999E+09]];
	LOCAL CONST Robtarget Tr_meulage_bavure_P117 :=[[-176.59375,-74.898296875,23],[0.675211408156727,-0.641835481352831,0.250443589204349,-0.263466843830552],[0,0,0,0],[8.999999E+09,8.999999E+09,8.999999E+09,8.999999E+09,8.999999E+09,8.999999E+09]];
	LOCAL CONST Robtarget Tr_meulage_bavure_P118 :=[[-172.119828125,-78.8538828125,23],[0.675391636342515,-0.641502769927745,0.250514068200051,-0.263748052822141],[0,0,0,0],[8.999999E+09,8.999999E+09,8.999999E+09,8.999999E+09,8.999999E+09,8.999999E+09]];
	LOCAL CONST Robtarget Tr_meulage_bavure_P119 :=[[-171.914234375,-79.1292890625,23],[0.675376040384996,-0.641009461244752,0.251033618538766,-0.264492338323684],[0,0,0,0],[8.999999E+09,8.999999E+09,8.999999E+09,8.999999E+09,8.999999E+09,8.999999E+09]];
	LOCAL CONST Robtarget Tr_meulage_bavure_P120 :=[[-171.673703125,-79.4758125,23],[0.67517404123548,-0.640361960984986,0.25197777200816,-0.265676072274146],[0,0,0,0],[8.999999E+09,8.999999E+09,8.999999E+09,8.999999E+09,8.999999E+09,8.999999E+09]];
	LOCAL CONST Robtarget Tr_meulage_bavure_P121 :=[[-170.833171875,-79.9912734375,23],[0.674790460030607,-0.639567544136697,0.253325912081974,-0.26727733500331],[0,0,0,0],[8.999999E+09,8.999999E+09,8.999999E+09,8.999999E+09,8.999999E+09,8.999999E+09]];
	LOCAL CONST Robtarget Tr_meulage_bavure_P122 :=[[-170.4779375,-80.325578125,23],[0.67423225661598,-0.638638374951426,0.255047931208165,-0.269262776789443],[0,0,0,0],[8.999999E+09,8.999999E+09,8.999999E+09,8.999999E+09,8.999999E+09,8.999999E+09]];
	LOCAL CONST Robtarget Tr_meulage_bavure_P123 :=[[-166.172609375,-84.645734375,23],[0.673514254235656,-0.637580329003595,0.257107603734907,-0.27159814710478],[0,0,0,0],[8.999999E+09,8.999999E+09,8.999999E+09,8.999999E+09,8.999999E+09,8.999999E+09]];
	LOCAL CONST Robtarget Tr_meulage_bavure_P124 :=[[-165.623765625,-85.4247890625,23],[0.672651364441619,-0.636416141116343,0.259452323342697,-0.274224596186207],[0,0,0,0],[8.999999E+09,8.999999E+09,8.999999E+09,8.999999E+09,8.999999E+09,8.999999E+09]];
	LOCAL CONST Robtarget Tr_meulage_bavure_P125 :=[[-162.01209375,-88.4931171875,23],[0.671665433778336,-0.635160654467858,0.262028242722515,-0.277087870718067],[0,0,0,0],[8.999999E+09,8.999999E+09,8.999999E+09,8.999999E+09,8.999999E+09,8.999999E+09]];
	LOCAL CONST Robtarget Tr_meulage_bavure_P126 :=[[-161.758609375,-88.7569921875,23],[0.670572036829874,-0.633835638502596,0.26478561921444,-0.280132294894868],[0,0,0,0],[8.999999E+09,8.999999E+09,8.999999E+09,8.999999E+09,8.999999E+09,8.999999E+09]];
	LOCAL CONST Robtarget Tr_meulage_bavure_P127 :=[[-161.430421875,-89.082796875,23],[0.669399576439395,-0.632463397803173,0.267658520247125,-0.283289911647313],[0,0,0,0],[8.999999E+09,8.999999E+09,8.999999E+09,8.999999E+09,8.999999E+09,8.999999E+09]];
	LOCAL CONST Robtarget Tr_meulage_bavure_P128 :=[[-159.816015625,-90.9409453125,23],[0.668183731128977,-0.631079475871746,0.27056246283204,-0.286470156027224],[0,0,0,0],[8.999999E+09,8.999999E+09,8.999999E+09,8.999999E+09,8.999999E+09,8.999999E+09]];
	LOCAL CONST Robtarget Tr_meulage_bavure_P129 :=[[-158.0838125,-93.0798046875,23],[0.666960416200685,-0.629722541997799,0.273414320010981,-0.289582342234762],[0,0,0,0],[8.999999E+09,8.999999E+09,8.999999E+09,8.999999E+09,8.999999E+09,8.999999E+09]];
	LOCAL CONST Robtarget Tr_meulage_bavure_P130 :=[[-157.573375,-93.738140625,23],[0.665777765500677,-0.62843183550617,0.276118213439555,-0.292527139414822],[0,0,0,0],[8.999999E+09,8.999999E+09,8.999999E+09,8.999999E+09,8.999999E+09,8.999999E+09]];
	LOCAL CONST Robtarget Tr_meulage_bavure_P131 :=[[-157.145671875,-94.4612890625,23],[0.664674000466626,-0.627245268825724,0.278596935525362,-0.295221261692505],[0,0,0,0],[8.999999E+09,8.999999E+09,8.999999E+09,8.999999E+09,8.999999E+09,8.999999E+09]];
	LOCAL CONST Robtarget Tr_meulage_bavure_P132 :=[[-157.058421875,-94.673015625,23],[0.663692749503011,-0.626206662176337,0.280764119687409,-0.297571268101035],[0,0,0,0],[8.999999E+09,8.999999E+09,8.999999E+09,8.999999E+09,8.999999E+09,8.999999E+09]];
	LOCAL CONST Robtarget Tr_meulage_bavure_P133 :=[[-156.769734375,-94.9203046875,23],[0.662875579599828,-0.625350693650194,0.282545738453429,-0.299500219704793],[0,0,0,0],[8.999999E+09,8.999999E+09,8.999999E+09,8.999999E+09,8.999999E+09,8.999999E+09]];
	LOCAL CONST Robtarget Tr_meulage_bavure_P134 :=[[-156.242375,-95.6268125,23],[0.662244092600293,-0.6247015735409,0.28390306424585,-0.300964708800475],[0,0,0,0],[8.999999E+09,8.999999E+09,8.999999E+09,8.999999E+09,8.999999E+09,8.999999E+09]];
	LOCAL CONST Robtarget Tr_meulage_bavure_P135 :=[[-152.299328125,-101.358796875,23],[0.661818711722511,-0.624279565337228,0.284800762117146,-0.301926386746523],[0,0,0,0],[8.999999E+09,8.999999E+09,8.999999E+09,8.999999E+09,8.999999E+09,8.999999E+09]];
	LOCAL CONST Robtarget Tr_meulage_bavure_P136 :=[[-148.09934375,-106.841765625,23],[0.661597111170914,-0.624078081802433,0.285252561877494,-0.302401696831258],[0,0,0,0],[8.999999E+09,8.999999E+09,8.999999E+09,8.999999E+09,8.999999E+09,8.999999E+09]];
	LOCAL CONST Robtarget Tr_meulage_bavure_P137 :=[[-146.512203125,-108.826234375,23],[0.661565316333922,-0.62408517069652,0.285288948126189,-0.302422300794347],[0,0,0,0],[8.999999E+09,8.999999E+09,8.999999E+09,8.999999E+09,8.999999E+09,8.999999E+09]];
	LOCAL CONST Robtarget Tr_meulage_bavure_P138 :=[[-145.057375,-110.472125,23],[0.66169847485193,-0.62427879048058,0.284960280429699,-0.302040988463753],[0,0,0,0],[8.999999E+09,8.999999E+09,8.999999E+09,8.999999E+09,8.999999E+09,8.999999E+09]];
	LOCAL CONST Robtarget Tr_meulage_bavure_P139 :=[[-144.42934375,-111.250765625,23],[0.661962151376284,-0.624626072921622,0.284336490479611,-0.301332273999205],[0,0,0,0],[8.999999E+09,8.999999E+09,8.999999E+09,8.999999E+09,8.999999E+09,8.999999E+09]];
	LOCAL CONST Robtarget Tr_meulage_bavure_P140 :=[[-143.793671875,-111.9365546875,23],[0.662318139747102,-0.625087624015738,0.283497099204904,-0.300382321062181],[0,0,0,0],[8.999999E+09,8.999999E+09,8.999999E+09,8.999999E+09,8.999999E+09,8.999999E+09]];
	LOCAL CONST Robtarget Tr_meulage_bavure_P141 :=[[-139.258453125,-116.6111328125,23],[0.662720811739723,-0.625626879633114,0.282529628332688,-0.299281042302664],[0,0,0,0],[8.999999E+09,8.999999E+09,8.999999E+09,8.999999E+09,8.999999E+09,8.999999E+09]];
	LOCAL CONST Robtarget Tr_meulage_bavure_P142 :=[[-134.7735625,-120.733734375,23],[0.663133201152644,-0.626203922928859,0.281513870501444,-0.298115657342667],[0,0,0,0],[8.999999E+09,8.999999E+09,8.999999E+09,8.999999E+09,8.999999E+09,8.999999E+09]];
	LOCAL CONST Robtarget Tr_meulage_bavure_P143 :=[[-134.4039375,-121.110828125,23],[0.663527962634208,-0.626793581897256,0.280506137456613,-0.296945711105713],[0,0,0,0],[8.999999E+09,8.999999E+09,8.999999E+09,8.999999E+09,8.999999E+09,8.999999E+09]];
	LOCAL CONST Robtarget Tr_meulage_bavure_P144 :=[[-133.9021875,-121.595125,23],[0.663875818473884,-0.627371547634675,0.27956568015543,-0.295832502175361],[0,0,0,0],[8.999999E+09,8.999999E+09,8.999999E+09,8.999999E+09,8.999999E+09,8.999999E+09]];
	LOCAL CONST Robtarget Tr_meulage_bavure_P145 :=[[-131.987640625,-123.5568828125,23],[0.664167378895508,-0.627924375771892,0.27871699354253,-0.294804186932895],[0,0,0,0],[8.999999E+09,8.999999E+09,8.999999E+09,8.999999E+09,8.999999E+09,8.999999E+09]];
	LOCAL CONST Robtarget Tr_meulage_bavure_P146 :=[[-128.20440625,-127.7205625,23],[0.664388012532047,-0.628436765970221,0.277993576513697,-0.29389687204482],[0,0,0,0],[8.999999E+09,8.999999E+09,8.999999E+09,8.999999E+09,8.999999E+09,8.999999E+09]];
	LOCAL CONST Robtarget Tr_meulage_bavure_P147 :=[[-126.3279453125,-129.7808671875,23],[0.66453950635694,-0.628914877191025,0.27738910527792,-0.293101699093997],[0,0,0,0],[8.999999E+09,8.999999E+09,8.999999E+09,8.999999E+09,8.999999E+09,8.999999E+09]];
	LOCAL CONST Robtarget Tr_meulage_bavure_P148 :=[[-124.547390625,-131.75534375,23],[0.664623442622356,-0.629355939003264,0.276904783791111,-0.292421822495732],[0,0,0,0],[8.999999E+09,8.999999E+09,8.999999E+09,8.999999E+09,8.999999E+09,8.999999E+09]];
	LOCAL CONST Robtarget Tr_meulage_bavure_P149 :=[[-122.425109375,-134.06734375,23],[0.664649393179945,-0.629765302885012,0.276523995887706,-0.291841270429622],[0,0,0,0],[8.999999E+09,8.999999E+09,8.999999E+09,8.999999E+09,8.999999E+09,8.999999E+09]];
	LOCAL CONST Robtarget Tr_meulage_bavure_P150 :=[[-117.879546875,-138.70953125,23],[0.664617657963224,-0.630150039787543,0.276240986027297,-0.291350671387426],[0,0,0,0],[8.999999E+09,8.999999E+09,8.999999E+09,8.999999E+09,8.999999E+09,8.999999E+09]];
	LOCAL CONST Robtarget Tr_meulage_bavure_P151 :=[[-114.123140625,-142.89259375,23],[0.664531844994589,-0.630508474990998,0.276052765555797,-0.290949068707239],[0,0,0,0],[8.999999E+09,8.999999E+09,8.999999E+09,8.999999E+09,8.999999E+09,8.999999E+09]];
	LOCAL CONST Robtarget Tr_meulage_bavure_P152 :=[[-113.915984375,-143.1503125,23],[0.664395945147682,-0.630846654098497,0.275949142288539,-0.290624496480027],[0,0,0,0],[8.999999E+09,8.999999E+09,8.999999E+09,8.999999E+09,8.999999E+09,8.999999E+09]];
	LOCAL CONST Robtarget Tr_meulage_bavure_P153 :=[[-113.854125,-143.20696875,23],[0.664208508723853,-0.631159545314825,0.275936660739697,-0.290385338053841],[0,0,0,0],[8.999999E+09,8.999999E+09,8.999999E+09,8.999999E+09,8.999999E+09,8.999999E+09]];
	LOCAL CONST Robtarget Tr_meulage_bavure_P154 :=[[-111.2149375,-145.93953125,23],[0.663973575113304,-0.631448876495812,0.2760085628058,-0.290225224922492],[0,0,0,0],[8.999999E+09,8.999999E+09,8.999999E+09,8.999999E+09,8.999999E+09,8.999999E+09]];
	LOCAL CONST Robtarget Tr_meulage_bavure_P155 :=[[-107.781828125,-149.4845625,23],[0.663686108896705,-0.631713478541125,0.276172832755231,-0.290150644209133],[0,0,0,0],[8.999999E+09,8.999999E+09,8.999999E+09,8.999999E+09,8.999999E+09,8.999999E+09]];
	LOCAL CONST Robtarget Tr_meulage_bavure_P156 :=[[-107.4350859375,-149.8185,23],[0.663347806837277,-0.631954018532913,0.276426641906932,-0.29015877940937],[0,0,0,0],[8.999999E+09,8.999999E+09,8.999999E+09,8.999999E+09,8.999999E+09,8.999999E+09]];
	LOCAL CONST Robtarget Tr_meulage_bavure_P157 :=[[-106.42696875,-150.885296875,23],[0.662969346075243,-0.632174474233761,0.276752029625922,-0.290233344724147],[0,0,0,0],[8.999999E+09,8.999999E+09,8.999999E+09,8.999999E+09,8.999999E+09,8.999999E+09]];
	LOCAL CONST Robtarget Tr_meulage_bavure_P158 :=[[-103.5145546875,-153.93065625,23],[0.662561281052729,-0.63238709356174,0.277124067789202,-0.29034697139503],[0,0,0,0],[8.999999E+09,8.999999E+09,8.999999E+09,8.999999E+09,8.999999E+09,8.999999E+09]];
	LOCAL CONST Robtarget Tr_meulage_bavure_P159 :=[[-101.476015625,-155.987890625,23],[0.662140987018903,-0.632605850143522,0.277507094551151,-0.290463361110491],[0,0,0,0],[8.999999E+09,8.999999E+09,8.999999E+09,8.999999E+09,8.999999E+09,8.999999E+09]];
	LOCAL CONST Robtarget Tr_meulage_bavure_P160 :=[[-99.91521875,-157.40284375,23],[0.661723175220867,-0.632848823830771,0.277865594160256,-0.290543485787572],[0,0,0,0],[8.999999E+09,8.999999E+09,8.999999E+09,8.999999E+09,8.999999E+09,8.999999E+09]];
	LOCAL CONST Robtarget Tr_meulage_bavure_P161 :=[[-95.1838046875,-162.357703125,23],[0.661328892842169,-0.633130699175647,0.278158394784154,-0.290546933669261],[0,0,0,0],[8.999999E+09,8.999999E+09,8.999999E+09,8.999999E+09,8.999999E+09,8.999999E+09]];
	LOCAL CONST Robtarget Tr_meulage_bavure_P162 :=[[-93.170046875,-164.57575,23],[0.660978318581272,-0.63347047947951,0.278341739880503,-0.290428459063105],[0,0,0,0],[8.999999E+09,8.999999E+09,8.999999E+09,8.999999E+09,8.999999E+09,8.999999E+09]];
	LOCAL CONST Robtarget Tr_meulage_bavure_P163 :=[[-92.8446328125,-164.96221875,23],[0.660685067813943,-0.63388082249735,0.278386019350301,-0.290157833373601],[0,0,0,0],[8.999999E+09,8.999999E+09,8.999999E+09,8.999999E+09,8.999999E+09,8.999999E+09]];
	LOCAL CONST Robtarget Tr_meulage_bavure_P164 :=[[-86.974734375,-172.471765625,23],[0.660448492958923,-0.634365331708519,0.278288454233532,-0.289730823895111],[0,0,0,0],[8.999999E+09,8.999999E+09,8.999999E+09,8.999999E+09,8.999999E+09,8.999999E+09]];
	LOCAL CONST Robtarget Tr_meulage_bavure_P165 :=[[-86.8349609375,-172.627109375,23],[0.660267443823802,-0.634912162235373,0.27806005310775,-0.289164409528043],[0,0,0,0],[8.999999E+09,8.999999E+09,8.999999E+09,8.999999E+09,8.999999E+09,8.999999E+09]];
	LOCAL CONST Robtarget Tr_meulage_bavure_P166 :=[[-85.0375703125,-174.592828125,23],[0.660129392967401,-0.635514201851154,0.277723111035527,-0.288480081431508],[0,0,0,0],[8.999999E+09,8.999999E+09,8.999999E+09,8.999999E+09,8.999999E+09,8.999999E+09]];
	LOCAL CONST Robtarget Tr_meulage_bavure_P167 :=[[-83.5334765625,-176.04225,23],[0.660008361859898,-0.636150305171494,0.277330637719802,-0.287731591743343],[0,0,0,0],[8.999999E+09,8.999999E+09,8.999999E+09,8.999999E+09,8.999999E+09,8.999999E+09]];
	LOCAL CONST Robtarget Tr_meulage_bavure_P168 :=[[-82.02225,-177.5301875,23],[0.659884628822309,-0.636791554301169,0.276934513874241,-0.286977469568576],[0,0,0,0],[8.999999E+09,8.999999E+09,8.999999E+09,8.999999E+09,8.999999E+09,8.999999E+09]];
	LOCAL CONST Robtarget Tr_meulage_bavure_P169 :=[[-81.117953125,-178.311359375,23],[0.65973211110143,-0.637416693835678,0.27658924740777,-0.286272402127147],[0,0,0,0],[8.999999E+09,8.999999E+09,8.999999E+09,8.999999E+09,8.999999E+09,8.999999E+09]];
	LOCAL CONST Robtarget Tr_meulage_bavure_P170 :=[[-77.3982265625,-181.77815625,23],[0.659527399767783,-0.637997409821093,0.276352580057264,-0.285678430254749],[0,0,0,0],[8.999999E+09,8.999999E+09,8.999999E+09,8.999999E+09,8.999999E+09,8.999999E+09]];
	LOCAL CONST Robtarget Tr_meulage_bavure_P171 :=[[-76.7605625,-182.352015625,23],[0.659250994193635,-0.638521111620716,0.276263327961345,-0.285232344402018],[0,0,0,0],[8.999999E+09,8.999999E+09,8.999999E+09,8.999999E+09,8.999999E+09,8.999999E+09]];
	LOCAL CONST Robtarget Tr_meulage_bavure_P172 :=[[-75.261625,-183.78846875,23],[0.658911194578663,-0.638988892595808,0.276309914071224,-0.284924664050088],[0,0,0,0],[8.999999E+09,8.999999E+09,8.999999E+09,8.999999E+09,8.999999E+09,8.999999E+09]];
	LOCAL CONST Robtarget Tr_meulage_bavure_P173 :=[[-71.51421875,-187.5036875,23],[0.658503692480433,-0.639389971476518,0.276508470307552,-0.284774326815237],[0,0,0,0],[8.999999E+09,8.999999E+09,8.999999E+09,8.999999E+09,8.999999E+09,8.999999E+09]];
	LOCAL CONST Robtarget Tr_meulage_bavure_P174 :=[[-69.8831484375,-189.33478125,23],[0.658037966511325,-0.639743858594419,0.276828742423399,-0.284744933912164],[0,0,0,0],[8.999999E+09,8.999999E+09,8.999999E+09,8.999999E+09,8.999999E+09,8.999999E+09]];
	LOCAL CONST Robtarget Tr_meulage_bavure_P175 :=[[-67.4805625,-192.29034375,23],[0.657546856302038,-0.640071000913404,0.277207344857509,-0.284775935630226],[0,0,0,0],[8.999999E+09,8.999999E+09,8.999999E+09,8.999999E+09,8.999999E+09,8.999999E+09]];
	LOCAL CONST Robtarget Tr_meulage_bavure_P176 :=[[-65.74346875,-194.3895625,23],[0.657055943343781,-0.640410816407022,0.277573691875675,-0.28478820046486],[0,0,0,0],[8.999999E+09,8.999999E+09,8.999999E+09,8.999999E+09,8.999999E+09,8.999999E+09]];
	LOCAL CONST Robtarget Tr_meulage_bavure_P177 :=[[-64.69805859375,-195.445703125,23],[0.656605526669167,-0.640789294747826,0.277849111676877,-0.284707100762275],[0,0,0,0],[8.999999E+09,8.999999E+09,8.999999E+09,8.999999E+09,8.999999E+09,8.999999E+09]];
	LOCAL CONST Robtarget Tr_meulage_bavure_P178 :=[[-63.16708203125,-197.107390625,23],[0.656243273443833,-0.641254120978163,0.277925057091266,-0.28442148482325],[0,0,0,0],[8.999999E+09,8.999999E+09,8.999999E+09,8.999999E+09,8.999999E+09,8.999999E+09]];
	LOCAL CONST Robtarget Tr_meulage_bavure_P179 :=[[-62.89013671875,-197.410640625,23],[0.656028426149213,-0.641865396803437,0.277664895615702,-0.283791688062345],[0,0,0,0],[8.999999E+09,8.999999E+09,8.999999E+09,8.999999E+09,8.999999E+09,8.999999E+09]];
	LOCAL CONST Robtarget Tr_meulage_bavure_P180 :=[[-62.745390625,-197.557296875,23],[0.656020921622686,-0.642675250403444,0.27693573292687,-0.282686527341594],[0,0,0,0],[8.999999E+09,8.999999E+09,8.999999E+09,8.999999E+09,8.999999E+09,8.999999E+09]];
	LOCAL CONST Robtarget Tr_meulage_bavure_P181 :=[[-61.5524609375,-198.78496875,23],[0.656303413509685,-0.643770437915633,0.275536415509512,-0.280900581006197],[0,0,0,0],[8.999999E+09,8.999999E+09,8.999999E+09,8.999999E+09,8.999999E+09,8.999999E+09]];
	LOCAL CONST Robtarget Tr_meulage_bavure_P182 :=[[-55.272765625,-205.282875,23],[0.656968392252936,-0.645236342700594,0.273242418421959,-0.27821066552861],[0,0,0,0],[8.999999E+09,8.999999E+09,8.999999E+09,8.999999E+09,8.999999E+09,8.999999E+09]];
	LOCAL CONST Robtarget Tr_meulage_bavure_P183 :=[[-53.76150390625,-206.848015625,23],[0.658112568173868,-0.647174873674862,0.269788327806151,-0.274347933608189],[0,0,0,0],[8.999999E+09,8.999999E+09,8.999999E+09,8.999999E+09,8.999999E+09,8.999999E+09]];
	LOCAL CONST Robtarget Tr_meulage_bavure_P184 :=[[-48.0354296875,-212.87246875,23],[0.659860289698431,-0.649700980366176,0.264823161486023,-0.268964174809361],[0,0,0,0],[8.999999E+09,8.999999E+09,8.999999E+09,8.999999E+09,8.999999E+09,8.999999E+09]];
	LOCAL CONST Robtarget Tr_meulage_bavure_P185 :=[[-45.6156015625,-215.4116875,23],[0.662327658927193,-0.652936972558167,0.257941668318395,-0.261651443396978],[0,0,0,0],[8.999999E+09,8.999999E+09,8.999999E+09,8.999999E+09,8.999999E+09,8.999999E+09]];
	LOCAL CONST Robtarget Tr_meulage_bavure_P186 :=[[-42.8251328125,-218.47553125,23],[0.665641790202712,-0.657007288032586,0.248623235890287,-0.251890684987035],[0,0,0,0],[8.999999E+09,8.999999E+09,8.999999E+09,8.999999E+09,8.999999E+09,8.999999E+09]];
	LOCAL CONST Robtarget Tr_meulage_bavure_P187 :=[[-39.6845390625,-222.010125,23],[0.66987584081194,-0.661990979481978,0.236321799840557,-0.239136588378081],[0,0,0,0],[8.999999E+09,8.999999E+09,8.999999E+09,8.999999E+09,8.999999E+09,8.999999E+09]];
	LOCAL CONST Robtarget Tr_meulage_bavure_P188 :=[[-38.00439453125,-224.01159375,23],[0.675062542016914,-0.667921826197803,0.220371354352097,-0.222727332483638],[0,0,0,0],[8.999999E+09,8.999999E+09,8.999999E+09,8.999999E+09,8.999999E+09,8.999999E+09]];
	LOCAL CONST Robtarget Tr_meulage_bavure_P189 :=[[-36.8472890625,-225.319484375,23],[0.681137457005554,-0.674729050060132,0.200035960427788,-0.201935851707147],[0,0,0,0],[8.999999E+09,8.999999E+09,8.999999E+09,8.999999E+09,8.999999E+09,8.999999E+09]];
	LOCAL CONST Robtarget Tr_meulage_bavure_P190 :=[[-35.7463671875,-226.562921875,23],[0.687846927287889,-0.682172787824729,0.174638800260325,-0.17609140131103],[0,0,0,0],[8.999999E+09,8.999999E+09,8.999999E+09,8.999999E+09,8.999999E+09,8.999999E+09]];
	LOCAL CONST Robtarget Tr_meulage_bavure_P191 :=[[-33.8753671875,-228.609296875,23],[0.694711263531949,-0.689774061905869,0.143686106400649,-0.144714569657453],[0,0,0,0],[8.999999E+09,8.999999E+09,8.999999E+09,8.999999E+09,8.999999E+09,8.999999E+09]];
	LOCAL CONST Robtarget Tr_meulage_bavure_P192 :=[[-33.3806171875,-229.09709375,23],[0.700983828295408,-0.696790441652343,0.107159048872046,-0.107803947678577],[0,0,0,0],[8.999999E+09,8.999999E+09,8.999999E+09,8.999999E+09,8.999999E+09,8.999999E+09]];
	LOCAL CONST Robtarget Tr_meulage_bavure_P193 :=[[-32.395751953125,-229.757140625,23],[0.705746273084166,-0.702308261787859,0.0657376997307427,-0.066059505647837],[0,0,0,0],[8.999999E+09,8.999999E+09,8.999999E+09,8.999999E+09,8.999999E+09,8.999999E+09]];
	LOCAL CONST Robtarget Tr_meulage_bavure_P194 :=[[-30.05749609375,-231.5466875,23],[0.708128455691908,-0.705449131690743,0.0211212892886218,-0.0212015087896238],[0,0,0,0],[8.999999E+09,8.999999E+09,8.999999E+09,8.999999E+09,8.999999E+09,8.999999E+09]];
	LOCAL CONST Robtarget Tr_meulage_bavure_P195 :=[[-27.008421875,-232.212671875,23],[0.707650490322343,-0.705727221979403,-0.0242555216855366,0.0243216235384146],[0,0,0,0],[8.999999E+09,8.999999E+09,8.999999E+09,8.999999E+09,8.999999E+09,8.999999E+09]];
	LOCAL CONST Robtarget Tr_meulage_bavure_P196 :=[[-26.4899296875,-232.26975,23],[0.704434037049025,-0.703261420338575,-0.0677522744924218,0.0678652445017855],[0,0,0,0],[8.999999E+09,8.999999E+09,8.999999E+09,8.999999E+09,8.999999E+09,8.999999E+09]];
	LOCAL CONST Robtarget Tr_meulage_bavure_P197 :=[[-26.11733984375,-232.165125,23],[0.699146022336523,-0.698692245152635,-0.107259119807064,0.107328781008645],[0,0,0,0],[8.999999E+09,8.999999E+09,8.999999E+09,8.999999E+09,8.999999E+09,8.999999E+09]];
	LOCAL CONST Robtarget Tr_meulage_bavure_P198 :=[[-24.48190234375,-231.5128125,23],[0.692676504046562,-0.692923853772991,-0.141545213080566,0.141494686360289],[0,0,0,0],[8.999999E+09,8.999999E+09,8.999999E+09,8.999999E+09,8.999999E+09,8.999999E+09]];
	LOCAL CONST Robtarget Tr_meulage_bavure_P199 :=[[-23.2855234375,-230.8535,23],[0.685851880516802,-0.686770279103938,-0.170339856629827,0.170112065928305],[0,0,0,0],[8.999999E+09,8.999999E+09,8.999999E+09,8.999999E+09,8.999999E+09,8.999999E+09]];
	LOCAL CONST Robtarget Tr_meulage_bavure_P200 :=[[-22.9039296875,-230.504859375,23],[0.679279964157993,-0.680840396215842,-0.193916549962972,0.19347210864781],[0,0,0,0],[8.999999E+09,8.999999E+09,8.999999E+09,8.999999E+09,8.999999E+09,8.999999E+09]];
	LOCAL CONST Robtarget Tr_meulage_bavure_P201 :=[[-20.74920703125,-228.30359375,23],[0.673316050619397,-0.675488356716607,-0.21289907873287,0.212214415611407],[0,0,0,0],[8.999999E+09,8.999999E+09,8.999999E+09,8.999999E+09,8.999999E+09,8.999999E+09]];
